FUNCTION_BLOCK "GCS7_E_Motor"	// FB 12
TITLE = Motor Control
//
//COPYRIGHT:    (C) 1996  BUHLER AG, CH-9240 UZWIL, SWITZERLAND
//
//PRODUCT:      GCS7
//
//TITLE:        Motor Control
//
//REVISION:     11  (GCPROVB)
//
//-------------------------------------------------------------------------
//
//IDENT:        AUTHOR:             DEPT:                       DATE:
//
//FB12.5.0      A. Egli             CT3                         13-Mar-2008
//              - OutpFaultReset 
//              (Software is compatible to 4.7 only GCPROVB has new revision)
//FB12.4.7      A. Egli             CT3                         04-Oct-2007
//              Interlocked Manual Mode: Use direction InOutManRev  
//FB12.4.6      A. Egli             CT3                         09-Mar-2005
//              StStopped--> StFault: Log Text 13 (not stopped)
//FB12.4.5      A. Egli             CT3                         26-Mar-2004
//              Manual Mode: Stop Motor when InHWStop or InDPFault
//FB12.4.4      A. Egli             CT3                         07-Nov-2003
//              Reset CmdOn, CmdNext when CmdOff
//FB12.4.3      A. Egli             CT3                         22-Aug-2003
//              No Start request  if InLocal
//FB12.4.2      A. Egli             CT3                         24-Jul-2003
//              Report: StStopped 
//FB12.4.1      A. Egli             CT3                         18-Jun-2003
//              Message Fault Started=Text Nr 11 
//FB12.4.0      A. Egli             CT3                         17-Jun-2002
//              New Release with one block 
//FB12.3.2      A.Egli              CT3                         22-Mai-2002
//              StStopped: Error 11: Fault stopping    
//FB12.3.1      A.Egli              CT3                         09-Nov-2001
//              Transition StStopping-->Starting in Local mode (InpFaultDev=0)    
//              Transition StStopping-->Stopped  in Local mode (InpFaultDev=1)    
//FB12.3.0      A.Egli              CT3                         28-Okt-2001
//              StCode 30: InpFaultDev=1 and InLocal=1              
//              StCode 31: InpFaultDev=1 and InLocal=0              
//FB12.2.11     A.Egli              CT3                         13-Mar-2001
//              Transition StStarting-->StFault in Local mode              
//FB12.2.10     A.Egli              CT3                         22-Jan-2001
//              Transition StStarting-->StFault after t0              
//              Interlocking PC Direct Control command with Gr.OutManualOff
//FB12.2.9      S. Kalberer         CT3                         28-Nov-2000
//              Condition for StStarting: No #tmpHeavyStartup (Netzwerk 8)      
//FB12.2.8      A. Egli             CT3                         24-Jul-2000
//              Local mode:  Transition Stopping -> Starting adapted
//FB12.2.7      S. Kalberer         CT3                         15-Mar-2000
//              Manual mode: Transition Stopping -> Starting adapted
//FB12.2.6      S. Kalberer         CT3                         02-Nov-1999
//              Count stopping time in StFault, StCode with InLocal adapted
//FB12.2E       S. Kalberer         CT3                         07-Apr-1999
//              Set outputs in StStarted Passive -> Active
//FB12.2D       A. Egli             CT3                         21-Dec-1998
//              StStopping by change speed if ParRestartDelay is true
//              Local mode: stay in StStopped if InpFaultDev = 1
//FB12.2C       A. Egli             CT3                         23-Nov-1998
//              InLocal; StStartedFdw or StStartedRev if input is set
//FB12.2B       A. Egli             CT3                         17-Jul-1998
//              Run Monitoring Time by changing speed
//FB12.2A       A. Egli             CT3                         04-Mai-1998
//              StFault = StCode 32
//FB12.1A       S. Kalberer         AEE61                       14-Jul-1997
//              1st Release in S7
//
//-------------------------------------------------------------------------
//
//PURPOSE:      MANUAL : see [MxxMAN]
//
//RESTRICTIONS: S7
//              ACCU2: Pointer to dynamic datas of the element
//              ACCU1: Pointer to parameter datas of the element
//              CmdOff, CmdOn: always active unless local mode
//
//-------------------------------------------------------------------------
//=======================================================
//Log Message: 
//------------------------------------------------------
// 0  stopped
// 2  started forward
// 5  started reverse
// 9  fault cancelled
//10  fault device
//11  fault running
//12  fault starting
//13  fault stopping
//
//=======================================================
//StCode:  State               
//------------------------------------------------------
//32 StFault+InpFaultDev=0     fault
//31 StFault+InpFaultDev=1     fault Device        (Active)
// 1 StStopped                 Stopped
//41 Stopped.HWStop            StStopped + InHWStop 
//51 Stopped.DPFault           StStopped + DPFault
//61 StStopped.FaultDev        StStopped + FaultDevice (Passiv)
// 2 StStarting                starting
// 3 StStartedFwdSlow          started forward slow
// 4 StStartedFwdFast          started forward fast
// 5 StStartedRevSlow          started reverse slow
// 6 StStartedRevFast          started reverse fast
// 7 StStopping                stopping
// 9 StStartRequest            StStopped+CmdNext
AUTHOR : EA
FAMILY : GCS7LL
NAME : Motor
VERSION : 5.0
VAR
  StCode : INT ;	//Element state code
  InEnableRev : BOOL ;	//Enable to run the element reverse
  InEnableFwd : BOOL ;	//Enable to run the element forward
  InSlow : BOOL ;	//Speed mode: 1= slow / 0= fast
  InpRunSlow : BOOL ;	//Digital input: 1= element is running slow
  InpRunFast : BOOL ;	//Digital input: 1= element is running fast
  InpRunRev : BOOL ;	//Digital input: 1= element is running reverse
  InpRunFwd : BOOL ;	//Digital input: 1= element is running forward
  InpFaultDev : BOOL ;	//Digital input: 1= overload or fault frequency converter
  CmdOff : BOOL ;	//Pulse to stop the element immediately (manual mode)
  CmdOn : BOOL ;	//Pulse to start the element immediately (manual mode)
  CmdNext : BOOL ;	//Pulse to start the element in automatic mode (see global flags)
  CmdFaultReset : BOOL ;	//Command to reset fault
  InLocal : BOOL ;	//1= Local mode (no fault by start with service switch)
  InManual : BOOL ;	//1= Manual/ 0=Automatic
  InReport : BOOL ;	//Report of all state transitions
  InSeqStop : BOOL ;	//Stop automatically after idling time
  InHWStop : BOOL ;	//HW stop is detected, no fault
  InDPFault : BOOL ;	//DP-Fault is detected, no fault
  OutIdling : BOOL ;	//Idling is active
  OutpRunSlow : BOOL ;	//Digital output to run slow
  OutpRunFast : BOOL ;	//Digital output to run fast
  OutpRunRev : BOOL ;	//Digital output to run reverse
  OutpRunFwd : BOOL ;	//Digital output to run forward
  OutpFaultReset : BOOL ;	//Reset Alarm (e.g.Softstart)
  StStopped : BOOL ;	//Element is stopped
  StStarting : BOOL ;	//Element is starting
  StStartedFwd : BOOL ;	//Element is started forward: Next element can start
  StStopping : BOOL ;	//Element is stopping
  StFault : BOOL ;	//Element has a fault
  StStartedRev : BOOL ;	//Element is started reverse: Next Element can start
  InOutManSlow : BOOL ;	//Manual speed mode: 1= slow / 0= fast
  InOutManRev : BOOL ;	//Manual direction mode: 1= reverse / 0= forward
  OutAlarmNrLog : INT ;	//Last textnumber send to log
  Par : STRUCT
   ParObjectNo : INT ;	//Is used for communication with PC, e.g. for message
   ParMsgType : INT ;	//Is used for message (translation of state)
   ParHornCode : INT ;	//Is used by horn module
   ParLogOff : BOOL ;	//Report is off
   ParManual : BOOL ;	//Manual mode without interlocking
   ParRestartDelay : BOOL ;	//No restart possible in StStopping
   Par2Speed : BOOL ;	//Element with 2 speeds
   ParHeavyStartup : BOOL ;	//Element with heavy startup
   spare45 : BOOL ;
   spare46 : BOOL ;
   OutEdgeFaultReset : BOOL ;	//Internal used
   OutDelayFault : BOOL ;	//Delay time is running: Changing speed
   OutFlagFaultDev : BOOL ;	//Flag InpFaultDev
   ParMonTime : INT ;	//After this time outputs must be equal inputs
   ParStartingTime : INT ;	//Delay time, until the element is ready to start production
   ParStoppingTime : INT ;	//Delay time, until the element has come to a standstill
   ParIdlingTime : INT ;	//Requested idling time to stop element in automatic mode
   ParDelayTime : INT ;	//Requested fault delay time by negative flag of input
   OutMonTime : INT ;	//Actual time: Monitoring
   OutTransitionTime : INT ;	//Actual time: Starting, stopping, change direction, idling
   OutDelayTime : INT ;	//Actual time: DelayTime
   InOutManPulseLen : INT ;	//Pulse length to start a the motor
  END_STRUCT ;
END_VAR
VAR_TEMP
  tmpLOGvalue : WORD ;	//LOG value
  tmpLenDyn : DINT ;
  tmpReport : BOOL ;	//Global LOG all
  tmpEnableRev : BOOL ;	//Global enable reverse
  tmpEnableFwd : BOOL ;	//Global enable forward
  tmpEnable : BOOL ;	//Global enable
  tmpSlow : BOOL ;	//Global slow speed flag
  tmpDelayOver : BOOL ;	//Delay time is over
  tmpMonOver : BOOL ;	//Monitoring time is over
  tmpTimeClear : BOOL ;	//Delay- and monitoring time must be cleared
  tmpStop : BOOL ;	//States to clear outputs
  tmpInpOutpDiff : BOOL ;	//Inpputs ar different to outputs
  tmpInpFault : BOOL ;	//Fault variable
  tmpInpRunSlow : BOOL ;	//Variable to simulate InpRunSlow
  tmpHeavyStartup : BOOL ;	//Any element is starting with HeavyStartup
  tmpLocal : BOOL ;
  tmpFaultDelayDone : BOOL ;
  tmpStarted : BOOL ;
END_VAR
BEGIN
NETWORK
TITLE =  Start Global
      L     34;
      T     #tmpLenDyn;	//--> Len dynamic data in byte
NETWORK
TITLE = PC Control
//=== Test Object number =====================
      L     "SYS_DirectCtrlDB".PC.ObjectNo;	//PCControl.ObjectNo
      L     #Par.ParObjectNo;	//Input ObjectNo
      <>I;
      JC    Ctrl;
//=== Test OType      ========================
      L     1012;	//Input object type
      L     "SYS_DirectCtrlDB".PC.ObjectType;	//PCControl.ObjectType
      <>I;
      JC    Ctrl;
//=== Test Handshake =========================
      A     "SYS_DirectCtrlDB".PC.Hsk.FExamine;	// Handshake.FExamine
      JC    pExa;
      A     "SYS_DirectCtrlDB".PC.Hsk.FDefineCmd;	// Handshake.FDefineCmd
      JC    pCmd;
      A     "SYS_DirectCtrlDB".PC.Hsk.FDefinePara;	// Handshake.FDefinePara
      JC    pPar;
pIni: L     2;	// FcInit
      UC    "SYS_DirectCtrl";
      JU    Ctrl;
// Write parameter 
pPar: LAR1  P#DBX 58.0;
      L     P##Par;
      L     DW#16#FFFFF;
      AD;
      +AR1;
      L     DBW [AR1,P#8.0];
      T     #Par.ParMonTime;
      L     DBW [AR1,P#10.0];
      T     #Par.ParStartingTime;
      L     DBW [AR1,P#12.0];
      T     #Par.ParStoppingTime;
      L     DBW [AR1,P#14.0];
      T     #Par.ParIdlingTime;
      L     DBW [AR1,P#16.0];
      T     #Par.ParDelayTime;
// Write new commands from PC to Interface object
pCmd: A     "SYS_DirectCtrlDB".PC.Cmd1[6];	// CmdManSlowOn
      AN    "GCS7_Gr_OutManualOff";	//Global.OutManualOff  [2.10]
      S     #InOutManSlow;
      A     "SYS_DirectCtrlDB".PC.Cmd1[7];	// CmdManRevOn;
      AN    "GCS7_Gr_OutManualOff";	//Global.OutManualOff  [2.10]
      S     #InOutManRev;
      A     "SYS_DirectCtrlDB".PC.Cmd1[8];	// CmdOff
      AN    "GCS7_Gr_OutManualOff";	//Global.OutManualOff  [2.10]
      S     #CmdOff;
      A     "SYS_DirectCtrlDB".PC.Cmd1[9];	// CmdOn
      AN    "GCS7_Gr_OutManualOff";	//Global.OutManualOff  [2.10]
      S     #CmdOn;
      A     "SYS_DirectCtrlDB".PC.Cmd1[10];	// CmdNext
      S     #CmdNext;
      A     "SYS_DirectCtrlDB".PC.Cmd1[11];	// CmdFaultReset
      S     #CmdFaultReset;
      A     "SYS_DirectCtrlDB".PC.Cmd1[13];	// CmdManualOn
      S     #InManual;
      A     "SYS_DirectCtrlDB".PC.Cmd1[14];	// CmdReportOn
      S     #InReport;
      A     "SYS_DirectCtrlDB".PC.Cmd2[6];	// CmdManSlowOff
      R     #InOutManSlow;
      A     "SYS_DirectCtrlDB".PC.Cmd2[7];	// CmdManRevOff;
      R     #InOutManRev;
      A     "SYS_DirectCtrlDB".PC.Cmd2[13];	// CmdManualOff
      R     #InManual;
      A     "SYS_DirectCtrlDB".PC.Cmd2[14];	// CmdReportOff
      R     #InReport;
      AN    "SYS_DirectCtrlDB".PC.Cmd1[1];	// CmdOnTickFwd
      O     "GCS7_Gr_OutManualOff";	//Global.OutManualOff
      JC    pIni;
      L     "SYS_DirectCtrlDB".PC.Cmd3;	// "SYS_PCControl".PC.Cmd3
      T     #Par.InOutManPulseLen;
      JU    pIni;
pExa: TAR2;	// Address Dynamic datas
      T     "SYS_DirectCtrlDB".GC.InDynAddr;	// -->PCControl.GC.InDynAddr
      L     #tmpLenDyn;	// Length Dynamic datas
      T     "SYS_DirectCtrlDB".GC.InDynLen;	// -->PCControl.GC.InDynLen
      L     0;
      T     "SYS_DirectCtrlDB".GC.InParaAddr;	// -->PCControl.GC.InParaAddr
      T     "SYS_DirectCtrlDB".GC.InParaLen;	// -->PCControl.GC.InParaLen
      L     1;	// Code FcExamine
      UC    "SYS_DirectCtrl";
      L     11;	//Revision
      T     "SYS_DirectCtrlDB".GC.Revision;
NETWORK
TITLE =  All State Init
//===Clear tmp Variable, when nessecary
Ctrl: CLR;
      =     #tmpTimeClear;
//===Global Group Orders===
      A     "GCS7_Gr_OutManualOn";	//Global.OutManualOn
      S     #InManual;
      A     "GCS7_Gr_OutManualOff";	//Global.OutManualOff
      R     #InManual;
      A     #InManual;
      S     "GCS7_Gr_InManual";	//Global.InManualMode
      AN    #InManual;
      A     #InLocal;
      =     #tmpLocal;
//---Report is on---
      O     "GCS7_Gr_OutReportAll";	//---Global OutReportAll
      O     #InReport;
      =     #tmpReport;
//---Heavy Startup---
      A     "GCS7_Gr_InHeavyStartup";	//---Global InHeavyStartup
      A     #Par.ParHeavyStartup;
      =     #tmpHeavyStartup;
//===Global Enable and Speed===
      A     #CmdOff;	//[4.4]
      R     #CmdOn;	//[4.4]
      R     #CmdNext;	//[4.4]
//---Enable / Manual No Interlocking Mode---
      AN    #InManual;
      JC    AUT;
      A(;	//[4.5]
      A     #InEnableFwd;
      AN    #InOutManRev;	//[4.7]
      AN    #Par.ParManual;
      O;
      AN    #InOutManRev;
      A     #Par.ParManual;
      );	//[4.5]
      AN    #InHWStop;	//[4.5]
      AN    #InDPFault;	//[4.5]
      =     #tmpEnableFwd;
      A(;	//[4.5]
      A     #InEnableRev;
      A     #InOutManRev;	//[4.7]
      AN    #Par.ParManual;
      O;
      A     #InOutManRev;
      A     #Par.ParManual;
      );	//[4.5]
      AN    #InHWStop;	//[4.5]
      AN    #InDPFault;	//[4.5]
      =     #tmpEnableRev;
//---Speed / Manual No Interlocking Mode---
      A     #InOutManSlow;
      ON    #Par.Par2Speed;
      =     #tmpSlow;
      JU    ENAB;
//---Enable / Automatic Interlocking Mode---
AUT:  A     #InEnableFwd;
      AN    #InHWStop;
      AN    #InDPFault;
      AN    #InLocal;
      =     #tmpEnableFwd;
      A     #InEnableRev;
      AN    #InHWStop;
      AN    #InDPFault;
      AN    #InLocal;
      =     #tmpEnableRev;
//---Speed / Automatic Interlocking Mode---
      A     #InSlow;
      ON    #Par.Par2Speed;
      =     #tmpSlow;
//---Enable / HardwareStop---
ENAB: X     #tmpEnableFwd;	//---Global Enable
      X     #tmpEnableRev;
      =     #tmpEnable;
//---For one speed, no Inp nessecary: Simulate InpRunSlow
      AN    #Par.Par2Speed;
      A     #OutpRunSlow;
      =     #tmpInpRunSlow;
// Check Input different to Output
      A     #InpRunFwd;
      X     #OutpRunFwd;
      O(;
      A     #InpRunRev;
      X     #OutpRunRev;
      );
      O(;
      A     #InpRunFast;
      X     #OutpRunFast;
      );
      O(;
      O     #InpRunSlow;
      O     #tmpInpRunSlow;
      X     #OutpRunSlow;
      );
      =     #tmpInpOutpDiff;
//---Both Inputs or InpFaultDevice active
      A     #InpRunFwd;	// local StStarting
      A     #InpRunRev;
      O;
      A     #InpRunSlow;	// local StStarting
      A     #InpRunFast;
      =     #tmpInpFault;
NETWORK
TITLE = Start as Pulse
      AN    #tmpEnable;
      ON    #InManual;
      O     #CmdOff;
      JC    STP1;
      L     0;
      L     #Par.InOutManPulseLen;
      >=I;
      JC    STP2;
      S     #CmdOn;
      AN    "GCS7_Gr_OutTick200ms";	// Decrement all 200ms
      JC    STP2;
      +     -2;
      T     #Par.InOutManPulseLen;
      L     0;
      >I;
      JC    STP2;
      S     #CmdOff;
STP1: L     0;
      T     #Par.InOutManPulseLen;
STP2: NOP   0;
NETWORK
TITLE = Fault delay time: ParDelayTime 
//Test or Running delay time ====================
//---Condition for Delay Fault
      AN    #tmpInpOutpDiff;
      AN    #InpFaultDev;
      O     #InHWStop;
      O     #InDPFault;
      JC    TFDO;
      A     #StStartedFwd;
      O     #StStartedRev;
      AN    #Par.OutDelayFault;
      O     #StStopped;
      A     #tmpInpOutpDiff;
      O     #InpFaultDev;
      JC    TFF1;
TFDO: R     #tmpFaultDelayDone;
      L     0;
      T     #Par.OutDelayTime;
      JU    TFF0;
TFF1: AN    "GCS7_Gr_OutTick200ms";	// Decrement all 200ms
      L     #Par.OutDelayTime;
      JC    TFF3;
      +     2;
TFF3: T     #Par.OutDelayTime;
      L     #Par.ParDelayTime;
      >=I;
      =     #tmpFaultDelayDone;
      JCN   TFF0;
      T     #Par.OutDelayTime;
TFF0: NOP   0;
NETWORK
TITLE = States
      O     #StStartedFwd;
      O     #StStartedRev;
      =     #tmpStarted;
      A     #StStopped;	//===State machine===
      JC    S0;
      O     #StStartedFwd;
      O     #StStartedRev;
      JC    S2;
      A     #StStopping;
      JC    S3;
      A     #StStarting;
      JC    S1;
      A     #StFault;
      JC    S4;
      S     #StStopped;	//Initialise: goto StStopped
NETWORK
TITLE = StStopped
//---Condition for StFault
S0:   A     #tmpFaultDelayDone;	// [4.0]
      O     #tmpInpFault;
      AN    #tmpLocal;	//2D:
      JC    S0S4;
//---Condition for StStarting: local
      AN    #tmpLocal;
      JC    S0J1;
      X     #InpRunFwd;
      X     #InpRunRev;
      JC    S0S1;
      JU    SAVE;
//---Condition for StStopped
S0J1: O     #CmdOff;
      ON    #tmpEnable;
      JC    SAVE;
//---Condition for StStarting: automatic
      O     #CmdNext;
      O     #CmdOn;
      AN    #InManual;
      AN    #InSeqStop;
      AN    #tmpHeavyStartup;
      JC    S0S1;
//---Condition for StStarting: manual 
      A     #InManual;
      A     #CmdOn;
      JCN   SAVE;
//---Transition -> StStarting
S0S1: R     #StStopped;
      JU    xxS1;
//---Transition -> StFault
S0S4: R     #StStopped;
      R     #tmpEnable;	//[4.6]
      JU    xxS4;
NETWORK
TITLE = StStarting
//== Any transition to StStarting
xxS1: SET;
      S     #StStarting;
      L     #Par.ParMonTime;	// Set actual vaule of timer
      T     #Par.OutMonTime;
      L     #Par.ParStartingTime;
      T     #Par.OutTransitionTime;
      A     #tmpLocal;	// No output set in local mode
      JC    SAVE;
      A     #Par.ParHeavyStartup;	// Set Global InHeavyStartup
      S     "GCS7_Gr_InHeavyStartup";
      A     #tmpEnableFwd;	// Set direction
      =     #OutpRunFwd;
      A     #tmpEnableRev;
      =     #OutpRunRev;
      A     #tmpSlow;	// Set speed
      =     #OutpRunSlow;
      NOT;
      =     #OutpRunFast;
      JU    SAVE;
//== Logic ====
//---Condition for StFault
S1:   A     #tmpInpFault;
      O     #tmpFaultDelayDone;	// [4.0]
      AN    #tmpLocal;
      JC    S1S4;
//---Condition for StStopped  local mode
      AN    #tmpLocal;
      JC    S11;
      A     #InpRunRev;
      XN    #InpRunFwd;
      JC    S1S3;
      JU    S12;
//---Condition for StStopped  other modes
S11:  ON    #tmpEnable;
      O     #CmdOff;
      O;
      A     #InSeqStop;
      AN    #InManual;
      O;
      AN    #OutpRunFwd;
      AN    #OutpRunRev;
      JC    S1S3;
//---Condition for StStarting
S12:  AN    "GCS7_Gr_OutTick200ms";
      L     #Par.OutTransitionTime;	// Set Timer 
      JC    S13;
      L     #Par.OutMonTime;
      +     -2;
      T     #Par.OutMonTime;
      L     #Par.OutTransitionTime;
      +     -2;
      T     #Par.OutTransitionTime;
S13:  L     0;
      <=I;	//---Condition for StStarted
      =     #tmpDelayOver;	// Starting time over
      A     #tmpDelayOver;	// Started forward
      A     #tmpEnableFwd;
      AN    #tmpInpOutpDiff;
      O;
      A     #tmpDelayOver;	// Started forward local  
      A     #InpRunFwd;
      A     #tmpLocal;
      JC    S1S2;
      A     #tmpDelayOver;	// Started reverse
      A     #tmpEnableRev;
      AN    #tmpInpOutpDiff;
      O;
      A     #tmpDelayOver;	// Started reverse local  
      A     #InpRunRev;
      A     #tmpLocal;
      JC    S15;
      L     #Par.OutMonTime;	//---Condition for StFault
      L     0;	// Monitoring time over
      <=I;
//      U     #tmpDelayOver; // Starting time over [2.10]
      AN    #tmpLocal;	//[2.11]
      A     #tmpInpOutpDiff;	// Inp not equal Outp
      JC    S1S4;
      JU    SAVE;
S1S2: R     #StStarting;	//---Transition -> StStartedFwd
      S     #StStartedFwd;
      S     #tmpTimeClear;	// Reset actual timer value
      A     #tmpHeavyStartup;	// Clear Global InHeavyStartup
      R     "GCS7_Gr_InHeavyStartup";
      JU    LOG1;
S15:  R     #StStarting;	//---Transition -> StStartedRev
      S     #StStartedRev;
      S     #tmpTimeClear;	// Reset actual timer value
      A     #tmpHeavyStartup;	// Clear Global InHeavyStartup
      R     "GCS7_Gr_InHeavyStartup";
      JU    LOG1;
//---Transition -> StStopping
S1S3: R     #StStarting;
      A     #tmpHeavyStartup;	// Clear Global InHeavyStartup
      R     "GCS7_Gr_InHeavyStartup";
      JU    xxS3;
//---Transition -> StFault
S1S4: R     #StStarting;
      A     #tmpHeavyStartup;	// Clear Global InHeavyStartup
      R     "GCS7_Gr_InHeavyStartup";
      JU    xxS4;
NETWORK
TITLE = StStarted
S2:   A     #tmpInpFault;	//---Condition for StFault
      O     #tmpFaultDelayDone;	// [4.0]
      AN    #tmpLocal;
      JC    S2S4;
//---Condition for StStopping: local mode
      AN    #tmpLocal;
      JC    S2J1;	// no speed changing and no idling 
      A     #StStartedFwd;	// Input Fwd goes off
      AN    #InpRunFwd;
      O;
      A     #StStartedRev;	// Input Rev goes off
      AN    #InpRunRev;
      JC    S2S3;
      JU    SAVE;
//---Condition for StStopping: autmatic
S2J1: A     #Par.Par2Speed;	//[Rel 2D -->
      A     #Par.ParRestartDelay;
      A     #tmpSlow;
      AN    #OutpRunSlow;
      O;
      A     #Par.Par2Speed;
      A     #Par.ParRestartDelay;
      AN    #tmpSlow;
      A     #OutpRunSlow;
      JC    S2S3;	// Condition for StStoppping  Rel 2D <--]
      ON    #tmpEnable;	// other modes
      O     #CmdOff;
      O;
      A     #OutpRunFwd;	// Change direction: Fwd --> Rev
      A     #tmpEnableRev;
      O;
      A     #OutpRunRev;	// Change direction: Rev --> Fwd
      A     #tmpEnableFwd;
      JC    S2S3;
//2E:---Condition for StStarted: set direction outputs
      A     #tmpEnableFwd;
      =     #OutpRunFwd;
      A     #tmpEnableRev;
      =     #OutpRunRev;
//---Condition for StStarted: speed changing
      A     #OutpRunSlow;
      AN    #tmpSlow;
      A     #Par.Par2Speed;	// Doubt only one speed
      AN    #Par.OutDelayFault;
      O;
      A     #OutpRunFast;	//---Condition for StStarted: speed changing
      A     #tmpSlow;
      A     #Par.Par2Speed;	// Doubt only one speed
      AN    #Par.OutDelayFault;
      JCN   S2F1;
      S     #Par.OutDelayFault;
      L     #Par.ParMonTime;
      L     #Par.ParDelayTime;
      <=I;
      JC    S2F2;
      L     #Par.ParMonTime;
S2F2: T     #Par.OutMonTime;
      JU    SAVE;
S2F1: A     #InpRunSlow;
      O     #InpRunFast;
      ON    #Par.Par2Speed;	// Doubt only one speed
      JC    S2J2;
      A     #tmpSlow;	// Set speed
      =     #OutpRunSlow;
      NOT;
      =     #OutpRunFast;
//Test or Running delay time ====================
S2J2: A     #tmpInpOutpDiff;	//---Condition for Delay Fault
      A     #Par.OutDelayFault;	// Set OutDelayFault Bit
      JC    S2T1;
      A     #InpRunFast;
      O     #InpRunSlow;
      ON    #Par.Par2Speed;	// Doubt only one speed
      A     #Par.OutDelayFault;
      JCN   S2J3;	// Check Idling
      R     #Par.OutDelayFault;
      S     #tmpTimeClear;
      JU    SAVE;
S2T1: AN    "GCS7_Gr_OutTick200ms";	// Decrement all 200ms
      L     #Par.OutMonTime;
      JC    S2T3;
      +     -2;
      T     #Par.OutMonTime;
S2T3: L     0;
      <=I;
      R     #Par.OutDelayFault;
      JCN   SAVE;
      A     #tmpEnable;	// Condition for StFault
      JC    S2S4;
      JU    S2S3;	// Condition for StStoppping
//---Idling time ----------------------
S2J3: O     #InSeqStop;
      ON    #OutIdling;	// Condition to reset Idling-Time
      JC    S2I1;
      R     #OutIdling;
      S     #tmpTimeClear;	// Reset actual timer value
      JU    SAVE;
S2I1: ON    #InSeqStop;	// Idling time active ?
      O     #InManual;
      JC    SAVE;
      A     #OutIdling;
      JC    S2I2;
      S     #OutIdling;	// Preset Idling Time
      L     #Par.ParIdlingTime;
      T     #Par.OutTransitionTime;
S2I2: AN    "GCS7_Gr_OutTick200ms";	// Set Idling Time
      L     #Par.OutTransitionTime;
      JC    S2I3;
      +     -2;
      T     #Par.OutTransitionTime;
S2I3: L     0;
      >I;	// Idling time over
      JC    SAVE;
S2S3: R     #StStartedFwd;	//---Transition -> StStopping
      R     #StStartedRev;
      R     #Par.OutDelayFault;
      JU    xxS3;
S2S4: R     #StStartedFwd;	//---Transition -> StFault
      R     #StStartedRev;
      R     #Par.OutDelayFault;
      R     #OutIdling;
      JU    xxS4;
NETWORK
TITLE = StStopping
//===Any transition to StStopping
xxS3: SET;
      S     #StStopping;
      R     #OutIdling;
      L     #Par.ParMonTime;	// Set monitoring time
      T     #Par.OutMonTime;
      L     #Par.ParStoppingTime;	// Set stopping time
      T     #Par.OutTransitionTime;
      JU    SAVE;
//===Logic =======================
//---Condition for StFault
S3:   A     #tmpInpFault;
      O     #tmpFaultDelayDone;	// [4.0]
      AN    #tmpLocal;	//[2.8] 
      JC    S3S4;
//---Condition for StStarting in InLocal
//[3.1]      U     #tmpInpFault                //[2.8]
//[3.1]      U     #tmpLocal                   //[2.8] 
//[3.1]      SPB   SAVE                        //[2.8]  
      X     #InpRunFwd;	//[2.8]
      X     #InpRunRev;	//[2.8]
      AN    #tmpInpFault;	//[3.1]
      A     #tmpLocal;	//[2.8] 
      JC    S3S1;	//[2.8] Transition -> StStarting 
//---Condition for StStarting: no Restart
      A     #Par.ParRestartDelay;
      O     #tmpHeavyStartup;	//[2.9]
      JC    S3J2;
      O     #CmdNext;	// automatic StStarting
      O     #CmdOn;
      AN    #InManual;
      AN    #InSeqStop;
      A     #tmpEnable;
      AN    #tmpLocal;	//[3.1] 
      JC    S3S1;
      A     #InManual;	// manual StStarting
      A     #CmdOn;
      A     #tmpEnable;	// [2.7]
      JC    S3S1;
//---Condition for StStopping
S3J2: AN    "GCS7_Gr_OutTick200ms";
      L     #Par.OutTransitionTime;	// Set Timer 
      JC    S3J3;
      L     #Par.OutMonTime;	//---Condition for StStopped
      +     -2;	// Set actual timer
      T     #Par.OutMonTime;
      L     #Par.OutTransitionTime;
      +     -2;
      T     #Par.OutTransitionTime;
S3J3: L     0;
      <=I;	// Stopping time over
      =     #tmpDelayOver;
      A     #tmpDelayOver;	// Stopped
      AN    #tmpInpOutpDiff;	// Inp equal Outp
      JC    S3S0;
      L     #Par.OutMonTime;
      L     0;	// Monitoring time over
      <=I;
      =     #tmpMonOver;
      A     #tmpMonOver;
      A     #tmpDelayOver;	// Stopping time over
      AN    #tmpInpOutpDiff;	// Inp equal Outp
      JC    S3S0;
      A     #tmpMonOver;	//---Condition for StFault
      A     #tmpInpOutpDiff;
      O;
      A     #tmpMonOver;
      A     #tmpDelayOver;
      A     #tmpInpOutpDiff;
      JCN   SAVE;
//---Transtition -> StFault
S3S4: R     #StStopping;
      JU    xxS4;
//---Transition -> StStarting
S3S1: R     #StStopping;
      JU    xxS1;
//---Transition -> StStopped
S3S0: R     #StStopping;
      S     #StStopped;
      S     #tmpTimeClear;	// Reset actual timer value
      JU    LOG1;
NETWORK
TITLE =  StFault
// Any transiton to Fault  
xxS4: SET;
      S     #StFault;
      S     "GCS7_Gr_InFaultFlag";	// Global.InFaultFlag
//    S     #tmpTimeClear               // Reset actual timer value
      CALL  "SYS_Horn_Code" (
           FcCode                   := 1,
           ParObjectType            := 1012,
           ParObjectNo              := #Par.ParObjectNo,
           ParHornCode              := #Par.ParHornCode);
      L     0;	//2.6
      T     #Par.OutMonTime;
      L     #Par.ParStoppingTime;
      T     #Par.OutTransitionTime;
      SET;
S4S4: JU    LOG4;
//===logic
S4:   L     0;	//---Condition to count stopping time
      L     #Par.OutTransitionTime;	// Set Timer 
      >=I;
      ON    "GCS7_Gr_OutTick200ms";
      JC    S4J1;
      +     -2;
      T     #Par.OutTransitionTime;
S4J1: A     #InpFaultDev;
      A     #tmpFaultDelayDone;	// [4.0]
      AN    #tmpLocal;
      FP    #Par.OutFlagFaultDev;
      JC    S4S4;
      AN    #CmdFaultReset;	//---Condition for StFault
      AN    "GCS7_Gr_OutFaultReset";	// OutFaultReset
      AN    #tmpLocal;
      JC    SAVE;
      A     #InpFaultDev;	//---Condition for StFault with LOG
      O     #tmpInpFault;	// MessageClass Error Fault stopping
      O     #tmpInpOutpDiff;
      AN    #tmpLocal;
      JC    S4S4;
      R     #StFault;	//---Transition -> StStopping
      S     #StStopping;
      R     #OutIdling;
      L     #Par.ParMonTime;	// Set monitoring time
      T     #Par.OutMonTime;
      JU    LOG9;
NETWORK
TITLE = LOG Message
//LOG transition to StStopped,StStartedXxx
LOG1: AN    #tmpReport;	// ReportAll?
      JC    SAVE;
      A     #StStartedFwd;
      L     B#(4, 2);	// MessageClass Info started fwd
      JC    LOG;
      A     #StStartedRev;
      L     B#(4, 5);	// MessageClass Info started rev
      JC    LOG;
      A     #StStopped;
      L     B#(4, 0);	// MessageClass Info stopped
      JC    LOG;	// [4.2]
      JU    SAVE;
//LOG transition to fault
LOG4: A     #InpFaultDev;
      =     #Par.OutFlagFaultDev;	//[4.0]
      L     B#(1, 10);	// MessageClass Error fault device
      JC    LOG;
      A     #tmpStarted;
      L     B#(1, 11);	// MessageClass Error fault started
      JC    LOG;
      AN    #tmpEnable;	//Fault Stopping
      L     B#(1, 13);
      JC    LOG;
      L     B#(1, 12);	// MessageClass Error fault starting
      JU    LOG;
//Log fault cancelled
LOG9: L     B#(3, 9);	// MessageClass Operater "fault cancelled"
LOG:  A     #Par.ParLogOff;	//---Set LOG Message
      JC    SAVE;
      T     #tmpLOGvalue;
      L     W#16#FF;
      AW;
      T     #OutAlarmNrLog;
      CALL  "GCS7_LogConvert" (
           ObjectNo                 := #Par.ParObjectNo,
           MsgType                  := #Par.ParMsgType,
           ClassMsgTxt              := #tmpLOGvalue,
           OType                    := 1012);	// LOG Message Converter / Entry / Contains Class and TextNo
NETWORK
TITLE = State Code
//--Stopped, Substate ---
SAVE: AN    #StStopped;
      JC    STC2;
      L     41;	//Code: StStopped.HWStop
      A     #InHWStop;
      JC    STC9;
      L     51;	//Code: StStopped.DPFault
      A     #InDPFault;
      JC    STC9;
      A     #InpFaultDev;	// 
      L     30;	//Code: StStopped.InpFaultDev
      JC    STC9;	// 
      A     #CmdNext;
      AN    #tmpLocal;	//[4.3]
      L     9;	// Code: starting requested
      JC    STC9;
      L     1;	// Code: stopped
      JC    STC9;
//--------------------
STC2: A     #StStarting;
      L     2;	// Code: starting
      JC    STC9;
      AN    #StStartedFwd;
      JC    STC3;
      L     3;	// 2.6 Code: started forward slow
      A     #InLocal;
      A     #InpRunSlow;
      O     #OutpRunSlow;
      ON    #Par.Par2Speed;
      JC    STC9;
      L     4;	// Code: started forward fast
      JU    STC9;
//--------------------
STC3: AN    #StStartedRev;
      JC    STC4;
      L     5;	// 2.6: Code: started reverse slow
      A     #InLocal;
      A     #InpRunSlow;
      O     #OutpRunSlow;
      ON    #Par.Par2Speed;
      JC    STC9;
      L     6;	// Code: started reverse fast
      JU    STC9;
//--------------------
STC4: A     #StStopping;
      L     7;	// Code: stopping
      JC    STC9;
      A     #InpFaultDev;	// [3.0]
      L     31;	// [3.0]
      JC    STC9;	// [3.0]
      L     32;	// Code: fault
STC9: L     #StCode;	// Old state code
      TAK;
      T     #StCode;	// Save state code
      <>I;
      L     3;	// Load code for CBit methode
      CC    "SYS_CBitCtrl";
NETWORK
TITLE = Global End
      A     #CmdFaultReset;	//[5.0]
      S     #Par.OutEdgeFaultReset;	//[5.0]
      A     "GCS7_Gr_OutTick1s";	//[5.0]
      R     #OutpFaultReset;	//[5.0]
      A     "GCS7_Gr_OutTick1s";	//[5.0]
      A     #Par.OutEdgeFaultReset;	//[5.0]
      R     #Par.OutEdgeFaultReset;	//[5.0]
      S     #OutpFaultReset;	//[5.0]
//---Clear all commands
      CLR;
      =     #CmdOn;
      =     #CmdOff;
      =     #CmdNext;
      =     #CmdFaultReset;
      O     #StStopped;	//---Reset Hardware Outputs
      O     #StStopping;
      O     #StFault;
      =     #tmpStop;
      ON    #tmpEnableFwd;	// Output Forward
      O     #tmpStop;
      R     #OutpRunFwd;
      ON    #tmpEnableRev;	// Output Reverse
      O     #tmpStop;
      R     #OutpRunRev;
      ON    #tmpSlow;	// Output Slow
      O     #tmpStop;
      R     #OutpRunSlow;
      O     #tmpSlow;	// Output Fast
      O     #tmpStop;
      R     #OutpRunFast;
//--Output for group 
      AN    #InLocal;
      O     #InManual;
      A     #InDPFault;
      S     "GCS7_Gr_InDPFault";
      AN    #InLocal;
      O     #InManual;
      A     #InHWStop;
      S     "GCS7_Gr_InHWStop";
//---Reset actual timer values
      AN    #tmpTimeClear;
      BEC;
      L     0;
      T     #Par.OutMonTime;
      T     #Par.OutTransitionTime;
END_FUNCTION_BLOCK

FUNCTION_BLOCK "GCS7_E_ValveControl"	// FB 13
TITLE = ValveControl
//  
//COPYRIGHT:    (C) 1996  BUHLER AG, CH-9240 UZWIL, SWITZERLAND
//
//PRODUCT:      GCS7
//
//TITLE:        Valve Control with Limit Switch (VLS)
//
//-------------------------------------------------------------------------
//
//IDENT:        AUTHOR:             DEPT:                       DATE:
//
//FB13.4.6      A. Egli             CT3                         02-Dec-2004
//              PCD:Ignor CmdLN, CmdHN as con M12.4=1
//FB13.4.5      A. Egli             CT3                         26-Nov-2004
//              ParDelayTime always used also for InpFaultDev
//FB13.4.4      A. Egli             CT3                         28-Jun-2004
//              Init state after Download is StNoPosition
//FB13.4.3      A. Egli             CT3                         04-Sep-2003
//              InStopCTime, StCode=12, StCode=14
//FB13.4.2      A. Egli             CT3                         04-Sep-2003
//              Message Text: Fault opening =12, fault closing=11
//FB13.4.1      A. Egli             CT3                         16-Jun-2003
//              Store text number, when calling FC4 
//FB13.4.0      A. Egli             CT3                         17-Jun-2002
//              New Release with one block 
//FB13.2.8      A. Egli             CT3                         16-Mar-2002
//              Set minimum MonTime =0.3s
//FB13.2.7      A. Egli             CT3                         03-Jul-2001
//              Transition during fault delay time is running
//FB13.2.6      S. Kalberer         CT3                         30-May-2000
//              Local mode: InpLN+InpHN -> StNoPosition
//FB13.2.5      S. Kalberer         CT3                         15-Mar-2000
//              PulseValve: change direction with CmdLN/CmdHN corrected
//FB13.2.4      S. Kalberer         CT3                         25-Nov-1999
//              PulseValve: StopAndGo corrected
//FB13.2D       A. Egli             CT3                         11-Oct-1999
//              Remove flag 12.2 (Gr.OutNext)
//FB13.2C       S. Kalberer         CT3                         05-Mar-1999
//              Interlocked Manual Mode: StHN->StLN if InEnableHN=0
//FB13.2B       A. Egli             CT3                         09-Dec-1998
//              Automatic Fault reset if InLocal
//FB13.2A       A. Egli             CT3                         04-Mai-1998
//              StFault = StCode 32
//FB13.1B       A. Egli             AEE61                       4-Nov-1997
//              ParManual
//FB13.1A       S. Kalberer         AEE61                       4-Jul-1997
//              1st Release in S7
//
//-------------------------------------------------------------------------
//
//PURPOSE:      MANUAL : see [VLSxxMAN]
//
//RESTRICTIONS: S7
//              ACCU2: Pointer to dynamic datas of the element
//              ACCU1: Pointer to parameter datas of the element
//
//-------------------------------------------------------------------------
//=======================================================
//Log Message: 
//------------------------------------------------------
// 0  LN
// 2  HN
// 9  fault cancelled
//10  fault device
//11  fault LN
//12  fault HN
//13  fault no position
//
//=======================================================
//StCode:  State               
//------------------------------------------------------
//32   StFault                 
// 1   StLN                    
//41   StLN.HWStop             StLN + InHWStop
//51   StLN.DPFault            StLN + InDPFault
// 2   StCtoHN                 
//12   StCtoHN                 StCtoHN + InStopCTime
// 3   StHN                    
//43   StHN.HWStop             StHN + InHWStop
//53   StHN.DPFault            StHN + InDPFault
// 4   StCtoLN                 
//14   StCtoLN                 StCtoLN + InStopCTime
// 5   StNoPosition            
//45   StNoPosition.HWStop     StNoPosition + InHWStop
//55   StNoPosition.DPFault    StNoPosition + InDPFault
//
//
AUTHOR : EA
FAMILY : GCS7LL
NAME : VLS
VERSION : 4.6
VAR
  StCode : INT ;	//Element state code
  InEnableLN : BOOL ;	//Target position is LN
  InEnableHN : BOOL ;	//Target position is HN
  InStopCTime : BOOL ;	//Stop Monitoring Time in State StCToLN and StCToHN
  spare0203 : BOOL ;
  spare0204 : BOOL ;
  InpLN : BOOL ;	//Digital input: limit switch low  position (closed)
  InpHN : BOOL ;	//Digital input: limit switch high position (open)
  InpFaultDev : BOOL ;	//Digital input: fault device
  CmdLN : BOOL ;	//Pulse to set position LN (manual mode)
  CmdHN : BOOL ;	//Pulse to set position HN (manual mode)
  CmdNext : BOOL ;	//Open next element
  CmdFaultReset : BOOL ;	//Command to reset fault
  InLocal : BOOL ;	//1= Local mode (no fault by start with service switch)
  InManual : BOOL ;	//1= Manual/ 0= Automatic
  InReport : BOOL ;	//Report of all state transition
  InSeqStop : BOOL ;	//Stop automatically after idling time
  InHWStop : BOOL ;	//HW stop is detected, no fault
  InDPFault : BOOL ;	//DP-Fault is detected, no fault
  OutIdling : BOOL ;	//Idling time is running
  OutDelayFault : BOOL ;	//Delay time is running
  OutMonFault : BOOL ;	//Monitoring time is running
  OutpLN : BOOL ;	//Digital output: valve low  position (closed)
  OutpHN : BOOL ;	//Digital output: valve high position (open)
  spare0407 : BOOL ;
  StLN : BOOL ;	//Element is in position LN
  StCtoHN : BOOL ;	//Changing to position HN
  StHN : BOOL ;	//Element is in position HN
  StCtoLN : BOOL ;	//Changing to position LN
  StFault : BOOL ;	//Element has a fault (time-out by positioning)
  StNoPosition : BOOL ;	//Element is not in a final position (only in local mode)
  OutAlarmNrLog : INT ;	//Last textnumber send to log
  Par : STRUCT
   ParObjectNo : INT ;	//Is used for communication with PC, e.g. for message
   ParMsgType : INT ;	//Is used for message (translation of state)
   ParHornCode : INT ;	//Is used by horn module
   ParLogOff : BOOL ;	//Report is off
   ParManual : BOOL  := TRUE;	//No interlocking in manual mode
   ParPulseValve : BOOL ;	//Valves with pulse signal
   ParContValve : BOOL ;	//Valves with continuous signal
   ParManualFlap : BOOL ;	//Manual flap, no valves
   ParMonTime : INT ;	//After this time the element mus be in final position
   ParPulseTimeHN : INT ;	//Delay time, if arrive the position HN
   ParPulseTimeLN : INT ;	//Delay time, if arrive the position LN
   ParIdlingTime : INT ;	//Requested idling time to close valve in automatic mode
   ParDelayTime : INT ;	//Requested fault delay time by negative flag of input
   OutMonTime : INT ;	//Actual time: Monitoring
   OutTransitionTime : INT ;	//Actual time: Change to LN or HN
   OutDelayTime : INT ;	//Actual time: DelayTime
   InOutManPulseLen : INT ;	//Pulse length to Move to HN
  END_STRUCT ;
END_VAR
VAR_TEMP
  tmpLOGvalue : WORD ;	//LOG value
  tmpLenDyn : DINT ;
  tmpReport : BOOL ;	//Global LOG all
  tmpEnable : BOOL ;	//Global enable
  tmpInpOk : BOOL ;	//Input ok variable
  tmpDelayOver : BOOL ;	//Delay time is over
  tmpDelayClear : BOOL ;	//Delay time must be cleared
  tmpMonFault : BOOL ;	//Global monitor fault
  tmpMonOver : BOOL ;	//Monitoring time over
  tmpMonClear : BOOL ;	//Monitoring time must be cleared
  tmpNoMon : BOOL ;	//Monitoring not active
  tmpManStopGo : BOOL ;	//Condition for StopAndGo in manual mode
  tmpNext : BOOL ;	//Global next
  tmpInEnableLN : BOOL ;
  tmpInEnableHN : BOOL ;
  tmpLocalFault : BOOL ;
  tmpLocal : BOOL ;
END_VAR
BEGIN
NETWORK
TITLE =  Start Global
      L     34;
      T     #tmpLenDyn;	//--> Len dynamic data in byte
NETWORK
TITLE = PC Control
//=== Test Object number =====================
      L     "SYS_DirectCtrlDB".PC.ObjectNo;	//PCControl.ObjectNo
      L     #Par.ParObjectNo;	//Input ObjectNo
      <>I;
      JC    aEnd;
//===     Test OType      ========================
      L     1013;	//Input object type
      L     "SYS_DirectCtrlDB".PC.ObjectType;	//PCControl.ObjectType
      <>I;
      JC    aEnd;
//===     Test Handshake =========================
      A     "SYS_DirectCtrlDB".PC.Hsk.FExamine;	// Handshake.FExamine
      JC    aExa;
      A     "SYS_DirectCtrlDB".PC.Hsk.FDefineCmd;	// Handshake.FDefineCmd
      JC    aCmd;
      A     "SYS_DirectCtrlDB".PC.Hsk.FDefinePara;	// Handshake.FDefinePara
      JC    aPar;
aIni: L     2;	// FcInit
      UC    "SYS_DirectCtrl";
      JU    aEnd;
// Write Parameter
aPar: LAR1  P#DBX 58.0;
      L     P##Par;
      L     DW#16#FFFFF;
      AD;
      +AR1;
      L     DBW [AR1,P#8.0];
      T     #Par.ParMonTime;
      L     DBW [AR1,P#10.0];
      T     #Par.ParPulseTimeHN;
      L     DBW [AR1,P#12.0];
      T     #Par.ParPulseTimeLN;
      L     DBW [AR1,P#14.0];
      T     #Par.ParIdlingTime;
      L     DBW [AR1,P#16.0];
      T     #Par.ParDelayTime;
// Write new commands from PC to Interface object
aCmd: A     "SYS_DirectCtrlDB".PC.Cmd1[8];	// CmdLN
      AN    "GCS7_Gr_OutManualOff";	//Global.OutManualOff  [2.10]
      S     #CmdLN;
      A     "SYS_DirectCtrlDB".PC.Cmd1[9];	// CmdHN
      AN    "GCS7_Gr_OutManualOff";	//Global.OutManualOff  [2.10]
      S     #CmdHN;
      A     "SYS_DirectCtrlDB".PC.Cmd1[10];	// CmdNext
      S     #CmdNext;
      A     "SYS_DirectCtrlDB".PC.Cmd1[11];	// CmdFaultReset
      S     #CmdFaultReset;
      A     "SYS_DirectCtrlDB".PC.Cmd1[13];	// CmdManualOn
      S     #InManual;
      A     "SYS_DirectCtrlDB".PC.Cmd1[14];	// CmdReportOn
      S     #InReport;
      A     "SYS_DirectCtrlDB".PC.Cmd2[13];	// CmdManualOff
      R     #InManual;
      A     "SYS_DirectCtrlDB".PC.Cmd2[14];	// CmdReportOff
      R     #InReport;
      AN    "SYS_DirectCtrlDB".PC.Cmd1[1];	// CmdOnTick
      O     "GCS7_Gr_OutManualOff";	//Global.OutManualOff
      JC    aIni;
      L     "SYS_DirectCtrlDB".PC.Cmd3;	// "SYS_PCControl".PC.Cmd3
      T     #Par.InOutManPulseLen;
      JU    aIni;
aExa: TAR2;	// Address Dynamic datas
      T     "SYS_DirectCtrlDB".GC.InDynAddr;	// -->PCControl.GC.InDynAddr
      L     #tmpLenDyn;	// Length Dynamic datas
      T     "SYS_DirectCtrlDB".GC.InDynLen;	// -->PCControl.GC.InDynLen
      L     0;
      T     "SYS_DirectCtrlDB".GC.InParaAddr;	// -->PCControl.GC.InParaAddr
      T     "SYS_DirectCtrlDB".GC.InParaLen;	// -->PCControl.GC.InParaLen
      L     1;	// Code FcExamine
      UC    "SYS_DirectCtrl";
      L     10;	//Revision
      T     "SYS_DirectCtrlDB".GC.Revision;
aEnd: NOP   0;
NETWORK
TITLE =  All State Init
//===Clear tmp Variable
      CLR;
      =     #tmpDelayClear;
      =     #tmpMonClear;
      =     #tmpMonFault;
//Minimum monitoring time                                 
      L     #Par.ParMonTime;	//[2.8]
      L     3;	//[2.8
      >=I;	//[2.8
      JC    ini0;	//[2.8
      T     #Par.ParMonTime;	//[2.8
//===Global Group Orders===
ini0: A     "GCS7_Gr_OutManualOn";	//Gr.OutManualOn
      S     #InManual;
      A     "GCS7_Gr_OutManualOff";	//Gr.OutManualOff
      R     #InManual;
      A     #InManual;
      S     "GCS7_Gr_InManual";	//Gr.InManualMode
      A     #InLocal;
      AN    #InManual;
      =     #tmpLocalFault;	//[4.0]
      A     #tmpLocalFault;	//[4.0]
      O     #InHWStop;	//[4.0]
      O     #InDPFault;	//[4.0]
      =     #tmpLocal;
//---Report is on---
      O     "GCS7_Gr_OutReportAll";	//Gr.OutReportAll
      O     #InReport;
      =     #tmpReport;
NETWORK
TITLE = Start as Pulse
      ON    #InManual;
      O     #CmdLN;
      JC    STP1;
      L     0;
      L     #Par.InOutManPulseLen;
      >=I;
      JC    STP2;
      S     #CmdHN;
      AN    "GCS7_Gr_OutTick200ms";	// Decrement all 200ms
      JC    STP2;
      +     -2;
      T     #Par.InOutManPulseLen;
      L     0;
      >I;
      JC    STP2;
      S     #CmdLN;
STP1: L     0;
      T     #Par.InOutManPulseLen;
STP2: NOP   0;
NETWORK
TITLE = Global Orders Part.2
//===Global Group Orders===
      A     #InEnableLN;
      =     #tmpInEnableLN;
      A     #InEnableHN;
      =     #tmpInEnableHN;
      AN    #InManual;
      ON    #Par.ParManual;
      JC    inJ1;
      A     #StLN;	//---Manual mode without interlocking
      O     #StCtoLN;
      O     #StFault;
      O     #CmdLN;
      AN    #CmdHN;
      =     #tmpInEnableLN;
      A     #StHN;
      O     #StCtoHN;
      O     #CmdHN;
      AN    #CmdLN;	// [2.5]
      =     #tmpInEnableHN;
//---Enable---
inJ1: A     #tmpInEnableLN;	//---Global enable
      X     #tmpInEnableHN;
      =     #tmpEnable;
//---Next---
      O     #CmdNext;	//---automatic StCtoHN
      =     #tmpNext;
//---Input ok---
      A(;
      A     #StLN;	//---Check Input: LN
      A     #InpLN;
      AN    #InpHN;
      O;
      A     #StHN;	// HN
      A     #InpHN;
      AN    #InpLN;
      O;
      AN    #StLN;	//[4.5]
      AN    #StHN;	//[4.5]
      );
      AN    #InpFaultDev;	//[4.0]
      =     #tmpInpOk;
//---Manual StopAndGo---
      A     #CmdLN;
      A     #CmdHN;
      =     #tmpManStopGo;
NETWORK
TITLE = ParDelayTime [4.5]
      NOP   0;
//[4.5]--->
      AN    #tmpInpOk;
      AN    #tmpLocal;	//===No monitoring in local mode
      JC    DTJO;
//--Stop Delay Time Fault ---
      R     #OutDelayFault;
      R     #tmpDelayOver;
      L     #Par.ParDelayTime;
      T     #Par.OutDelayTime;
      JU    DTD9;
//--Run Delay Time Fault ---
DTJO: L     0;
      L     #Par.OutDelayTime;
      >=I;
      ON    "GCS7_Gr_OutTick200ms";	// Decrement all 200ms
      JC    DTD2;
      +     -2;
      T     #Par.OutDelayTime;
DTD2: L     0;
      <=I;
      =     #tmpDelayOver;
      >I;
      =     #OutDelayFault;
DTD9: NOP   0;
//<---[4.5]
NETWORK
TITLE = Monitoring
// Monitoring active only in states StCtoLN and StCtoHN.
// Every transition into these both states will refresh the monitoring time.
      A     #tmpLocal;	//===No monitoring in local mode
      JC    STAT;
//===Condition for not monitoring
      A     #StCtoLN;
      O     #StCtoHN;
      ON    #OutMonFault;	// Clear monitoring information
      JC    MON2;
      R     #OutMonFault;
      S     #tmpMonClear;	// Reset actual value of timer
MON2: AN    #OutMonFault;	//---Condition for monitoring
      JC    STAT;
      A     #InpLN;	// [4.3]
      O     #InpHN;	// [4.3]
      A     #InStopCTime;
      ON    "GCS7_Gr_OutTick200ms";	// Global Tick 200ms
      L     #Par.OutMonTime;
      JC    MO21;
      +     -2;	// Decrement all 200ms
      T     #Par.OutMonTime;
MO21: L     0;
      <=I;	// Check t4/t5 over
      R     #OutMonFault;	// Reset monitoring bits
      =     #tmpMonFault;	//---Condition for monitoring fault
NETWORK
TITLE = States
STAT: A     #StLN;	//===State machine===
      JC    LN;
      A     #StCtoHN;
      JC    CHN;
      A     #StHN;
      JC    HN;
      A     #StCtoLN;
      JC    CLN;
      A     #StNoPosition;
      JC    NPS;
      A     #StFault;
      JC    FLT;
//---Initialise if no state
      S     #StNoPosition;	//[4.4]
      JU    NPS;	//[4.4]  
NETWORK
TITLE = StLN
LN:   AN    #tmpLocal;	//---Condition for StNoPosition: local
      JC    LN1;
      A     #InHWStop;	//[4.0]
      O     #InDPFault;	//[4.0]
      JC    SAVE;	//[4.0]
      AN    #InpLN;
      O;	// [2.6]
      A     #InpLN;	// [2.6]
      A     #InpHN;	// [2.6]
      JC    TNPS;
      JU    SAVE;
LN1:  A     #Par.ParManualFlap;	//===Manual flap function
      AN    #tmpInpOk;	//  without checking t4
      A(;
      AN    #tmpEnable;	// in automatic mode check Enable
      AN    #InManual;
      O;
      A     #InManual;	// not in manual mode
      );
      JC    TCHN;
      A     #tmpDelayOver;	//[4.5] Condition for fault
      JC    LN9;
//===Pulse Valve and Manual Flap
      A     #Par.ParContValve;
      JC    LN3;
      A     #tmpNext;
      AN    #InManual;
      O     #CmdHN;
      A     #tmpInEnableHN;
      AN    #tmpInEnableLN;
      JC    TCHN;
      JU    SAVE;
//===Continuous Valve: automatic StCtoHN
LN3:  A     #tmpNext;
      AN    #InManual;
      AN    #InSeqStop;
      O     #CmdHN;
      A     #tmpInEnableHN;
      JC    TCHN;
      JU    SAVE;
LN9:  R     #StLN;	//---Transition -> StFault
      L     B#(1, 10);	// MessageClass Error fault device
      A     #InpFaultDev;
      JC    xxS4;
      L     B#(1, 11);	// MessageClass Error fault LN
      JU    xxS4;
NETWORK
TITLE = StCtoHN
//---Change into local mode
CHN:  AN    #tmpLocal;
      JC    CHN1;
      A     #InpLN;	// StLN
      AN    #InpHN;
      JC    TLN;
      A     #InpHN;	// StHN
      AN    #InpLN;
      JC    THN;
      JU    TNPS;	// NoPosition
//---Condition for StFault
CHN1: O     #tmpMonFault;
      O     #tmpDelayOver;	//[4.5]
      JC    CHN9;
//---Condition for Pulse Time: not local
      AN    #InpHN;
      O;
      A     #InpLN;
      A     #InpHN;
      JCN   CHD1;
      L     #Par.ParPulseTimeHN;	//[4.5]
      T     #Par.OutTransitionTime;	//[4.5]
      JU    CHN2;	//[4.5]
CHD1: AN    "GCS7_Gr_OutTick200ms";	// Decrement all 200ms
      L     #Par.OutTransitionTime;
      JC    CHD2;
      +     -2;
      T     #Par.OutTransitionTime;
CHD2: L     0;	// Condition for StHN;
      <=I;
      JC    THN;
CHN2: A     #Par.ParContValve;	//---Pulse time (t1) not over
      JC    CHN3;	//===Pulse Valve and Manual Flap
      A     #Par.ParManualFlap;	// Manual flap function
      A     #InpLN;	//  Input changes
      AN    #InpHN;
      AN    #tmpEnable;
      JC    TCLN;
//---Automatic/manual mode: -> StCtoLN
      A     #tmpNext;
      AN    #InManual;
      O     #CmdLN;
      A     #tmpInEnableLN;
      AN    #tmpInEnableHN;
      JC    TCLN;
      A     #Par.ParManualFlap;	// No StopAndGo with ManualFlap
      JC    SAVE;
      AN    #tmpEnable;	// StopAndGo -> StHN
      O     #tmpManStopGo;	// 2.4: CmdLN and CmdHN
      A     #InpHN;
      AN    #InpLN;
      JC    THN;
      AN    #tmpEnable;	// StopAndGo -> StLN
      O     #tmpManStopGo;	// 2.4: CmdLN and CmdHN
      A     #InpLN;
      AN    #InpHN;
      JC    TLN;
      AN    #tmpEnable;	// StopAndGo -> StNoPosition
      O     #tmpManStopGo;	// 2.4: CmdLN and CmdHN
      JC    TNPS;
      JU    SAVE;	// Condition for StCtoHN
//===Continuous Valve:manual StCtoLN      
CHN3: A     #InManual;	//---Manual mode: StCtoLN
      A     #CmdLN;
      ON    #tmpInEnableHN;	//2C:---Automatic + interlocked manual mode: StCtoLN
      O;
      A     #InSeqStop;	// idling activated?
      AN    #InManual;
      JC    TCLN;
      JU    SAVE;
//---Transition -> StFault
CHN9: R     #StCtoHN;
      L     B#(1, 10);	// MessageClass Error fault device
      A     #InpFaultDev;
      JC    xxS4;
      L     B#(1, 12);	// MessageClass Error fault LN      //[4.2]
      A     #InpLN;
      JC    xxS4;
      L     B#(1, 13);	// MessageClass Error fault no position
      JU    xxS4;
NETWORK
TITLE = StHN
HN:   AN    #tmpLocal;	//---Condition for StNoPosition: local
      JC    HN1;
      A     #InHWStop;
      O     #InDPFault;
      AN    #Par.ParContValve;
      JC    SAVE;
      AN    #InpHN;
      O;	// [2.6]
      A     #InpLN;	// [2.6]
      A     #InpHN;	// [2.6]
      JC    TNPS;
      JU    SAVE;
HN1:  A     #Par.ParManualFlap;	//===Hand manual flap function
      AN    #tmpInpOk;	//  without checking t4
      A(;
      AN    #tmpEnable;	// in automatic mode check Enable
      AN    #InManual;
      O;
      A     #InManual;	// not in manual mode
      );
      JC    TCLN;
      A     #tmpDelayOver;	//[4.5] Condition for fault
      JC    HN9;
//===Pulse Valve and Manual Flap
      A     #Par.ParContValve;	//---Input HN ok
      JC    HN3;
      A     #tmpNext;	//---automatic StCtoLN
      O     #CmdLN;
      A     #tmpInEnableLN;
      AN    #tmpInEnableHN;
      O;
      A     #InManual;	//---manual StCtoLN, only with Pulse Valve
      A     #CmdLN;
      AN    #tmpEnable;
      A     #Par.ParPulseValve;
      JC    TCLN;
      JU    SAVE;
//===Continuous Valve: manual StCtoLN
HN3:  A     #InManual;	//---Manual mode: StCtoLN
      A     #CmdLN;
      ON    #tmpInEnableHN;	//2C:---Automatic + interlocked manual mode: StCtoLN
      JC    TCLN;
      O     #InSeqStop;	//---Idling time  
      ON    #OutIdling;	// Condition to reset Idling-Time
      JC    HNI1;
      R     #OutIdling;
      JU    SAVE;
HNI1: ON    #InSeqStop;	// Idling time active ?
      O     #InManual;
      JC    SAVE;
      A     #OutIdling;
      JC    HNI2;
      S     #OutIdling;	// Preset Idling Time
      L     #Par.ParIdlingTime;
      T     #Par.OutTransitionTime;
HNI2: AN    "GCS7_Gr_OutTick200ms";	// Set Idling Time
      L     #Par.OutTransitionTime;
      JC    HNI3;
      +     -2;
      T     #Par.OutTransitionTime;
HNI3: L     0;
      <=I;	// Idling time over
      JC    TCLN;
      JU    SAVE;
HN9:  R     #StHN;	//---Transition -> StFault
      L     B#(1, 10);	// MessageClass Error fault device
      A     #InpFaultDev;
      JC    xxS4;
      L     B#(1, 12);	// MessageClass Error fault HN
      JU    xxS4;
NETWORK
TITLE = StCtoLN
//---Change into local mode ---
CLN:  AN    #tmpLocal;
      JC    CLN1;
      A     #InpLN;	// StLN
      AN    #InpHN;
      JC    TLN;
      A     #InpHN;	// StHN
      AN    #InpLN;
      JC    THN;
      JU    TNPS;	//--> StNoPosition
//---Condition for StFault
CLN1: O     #tmpMonFault;
      O     #tmpDelayOver;	//[4.5]
      JC    CLN9;
//---Condition for Pulse Time: not local---
      AN    #InpLN;
      O;
      A     #InpLN;
      A     #InpHN;
      JCN   CLD1;	//[4.5]
      L     #Par.ParPulseTimeLN;	//[4.5]
      T     #Par.OutTransitionTime;	//[4.5]
      JU    CLN2;
CLD1: AN    "GCS7_Gr_OutTick200ms";	// Decrement all 1s
      L     #Par.OutTransitionTime;
      JC    CLD2;
      +     -2;
      T     #Par.OutTransitionTime;
CLD2: L     0;	// Condition for StLN;
      <=I;
      JC    TLN;
CLN2: A     #Par.ParContValve;	//---Pulse time (t1) not over
      JC    CLN3;	//===Pulse Valve and Manual Flap
      A     #Par.ParManualFlap;	// Manual flap function
      A     #InpHN;	//  Input changes
      AN    #InpLN;
      AN    #tmpEnable;
      JC    TCHN;
      A     #tmpNext;	//-> StCtoHN
      AN    #InManual;
      O     #CmdHN;	//2.4: CmdLN -> CmdHN
      A     #tmpInEnableHN;
      AN    #tmpInEnableLN;
      JC    TCHN;
      A     #Par.ParManualFlap;	// No StopAndGo with ManualFlap
      JC    SAVE;
      AN    #tmpEnable;	//---StopAndGo: automatic StHN
      O     #tmpManStopGo;	// 2.4: CmdLN and CmdHN
      A     #InpHN;
      AN    #InpLN;
      JC    THN;
      AN    #tmpEnable;	// StopAndGo -> StLN
      O     #tmpManStopGo;	// 2.4: CmdLN and CmdHN
      A     #InpLN;
      AN    #InpHN;
      JC    TLN;
      AN    #tmpEnable;	// StopAndGo -> StNoPosition
      O     #tmpManStopGo;	// 2.4: CmdLN and CmdHN
      JC    TNPS;
      JU    SAVE;
//                                ===Continuous Valve
CLN3: A     #tmpNext;	//---automatic StCtoHN
      AN    #InManual;
      AN    #InSeqStop;
      O     #CmdHN;
      A     #tmpInEnableHN;
      JC    TCHN;
      JU    SAVE;
CLN9: R     #StCtoLN;	//---Transition -> StFault
      L     B#(1, 10);	// MessageClass Error fault device
      A     #InpFaultDev;
      JC    xxS4;
      L     B#(1, 11);	// MessageClass Error fault LN //[4.2]
      A     #InpHN;
      JC    xxS4;
      L     B#(1, 13);	// MessageClass Error fault no position
      JU    xxS4;
NETWORK
TITLE =  StNoPosition;
//Valid state for all valves in local mode
//  and in not local mode only for pulse valve and manual flap
NPS:  A     #InpLN;	// -> StLN
      AN    #InpHN;
      JC    TLN;
      A     #InpHN;	// -> StHN
      AN    #InpLN;
      JC    THN;
      A     #tmpLocal;
      JC    SAVE;
//===Manual and automatic mode: InpLN -> StCtoLN
      A     #tmpDelayOver;	//--Condition for StFault
      JC    NPS9;
      A     #Par.ParManualFlap;	//--Condition for StFault
      JC    NPSn;
      A     #tmpNext;	// -> StCtoHN
      AN    #InManual;
      O     #CmdHN;
      A     #tmpInEnableHN;
      AN    #tmpInEnableLN;
      JC    TCHN;
      A     #tmpNext;	// -> StCtoLN
      AN    #InManual;
      O     #CmdLN;
      A     #tmpInEnableLN;
      AN    #tmpInEnableHN;
      JC    TCLN;
      JU    SAVE;
NPS9: R     #StNoPosition;	//---Transition -> StFault
      L     B#(1, 10);	//MessageClass Error fault device
      JU    xxS4;
NPSn: R     #StNoPosition;	//---Transition -> StFault
      L     B#(1, 13);	//MessageClass Error fault no position
      JU    xxS4;
NETWORK
TITLE =  StFault
//Change state conditions
//-----------------------
//All valves:
//FaultReset -> InLocal     -> InpHN  --> StHN
//                             InpLN  --> StLN
//                             no Inp --> StNoPosition
//                             InpHN and InpLN --> StNoPosition
//           -> not InLocal -> InpHN and InpLN --> StFault (reLOG fault)
//
//Pulse valve and Manual flap:
//FaultReset -> not InLocal -> InpHN  --> StCtoHN (start monitoring)
//                             InpLN  --> StCtoLN (  "        "    )
//                             no Inp --> StNoPosition
//Continuous valve:
//FaultReset -> not InLocal -> InpHN  --> StFault (reLOG fault)
//                             InpLN  --> StCtoLN (start monitoring)
//                             no Inp --> StFault (reLOG fault)
xxS4: SET;
      S     #StFault;
      S     "GCS7_Gr_InFaultFlag";	// InFaultFlag
      S     #tmpMonClear;
      T     #tmpLOGvalue;	//[4.1]
      CALL  "SYS_Horn_Code" (
           FcCode                   := 1,
           ParObjectType            := 1013,
           ParObjectNo              := #Par.ParObjectNo,
           ParHornCode              := #Par.ParHornCode);
      L     #tmpLOGvalue;	//[4.1]
      JU    LOG;
//Logic
//Local
FLT:  AN    #tmpLocalFault;
      JC    FLT1;
      A     #InpHN;	// -> StHN
      AN    #InpLN;
      JC    FLT7;
      A     #InpLN;	// -> StLN
      AN    #InpHN;
      JC    FLT6;
      JU    FLT8;	// No Input -> StNoPosition
//Remote
FLT1: AN    #CmdFaultReset;	//---Condition for StFault
      AN    "GCS7_Gr_OutFaultReset";	// OutFaultReset
      JC    SAVE;
      A     #InpFaultDev;	//---Condition for StFault with LOG
      L     B#(1, 10);	// MessageClass Error fault device
      JC    LOG;
      A     #InpLN;	//===All valves: Both Inputs -> StFault
      A     #InpHN;
      L     B#(1, 13);	// MessageClass Error fault no position
      JC    LOG;
      A     #InpLN;	// Input LN -> StCtoLN
      JC    FLT4;
      A     #Par.ParContValve;
      JC    FLT2;	//---Pulse Valve and Manual Flap: not local
      A     #InpHN;	// -> StCtoHN
      JC    FLT5;
      JU    FLT8;	// No Input -> StNoPosition
FLT2: A     #InpHN;	//---Continuous valve
      L     B#(1, 11);	// MessageClass Error fault LN
      JC    LOG;
      L     B#(1, 13);	// MessageClass Error fault no position
      JU    LOG;
FLT4: S     #StCtoLN;	//---Transition -> StCtoLN
      S     #OutMonFault;	// Activate monitoring
      L     #Par.ParPulseTimeLN;
      T     #Par.OutTransitionTime;
      L     #Par.ParMonTime;
      T     #Par.OutMonTime;
      JU    FLM;
FLT5: S     #StCtoHN;	//---Transition -> StCtoHN
      S     #OutMonFault;	// Activate monitoring
      L     #Par.ParPulseTimeHN;
      T     #Par.OutTransitionTime;
      L     #Par.ParMonTime;
      T     #Par.OutMonTime;
      JU    FLM;
FLT6: S     #StLN;	//---Transition -> StLN
      JU    FLM;
FLT7: S     #StHN;	//---Transition -> StHN
      JU    FLM;
FLT8: S     #StNoPosition;	//---Transition -> StNoPosition
FLM:  R     #StFault;
      L     B#(3, 9);	// MessageClass Operate fault cancelled
      JU    LOG;
NETWORK
TITLE = General Transitions
TCLN: SET;	// set VKE=1
      R     #StHN;	//---Transition -> StCtoLN
      R     #StCtoHN;
      R     #StNoPosition;
      S     #StCtoLN;
      R     #OutIdling;
      S     #OutMonFault;	// Activate monitoring
      L     #Par.ParPulseTimeLN;	//[4.5]
      T     #Par.OutTransitionTime;	//[4.5]
      L     #Par.ParMonTime;
      T     #Par.OutMonTime;
      JU    SAVE;
TCHN: SET;	// set VKE=1
      R     #StLN;	//---Transition -> StCtoHN
      R     #StCtoLN;
      R     #StNoPosition;
      S     #StCtoHN;
      S     #OutMonFault;	// Activate monitoring
      L     #Par.ParPulseTimeHN;	//[4.5]
      T     #Par.OutTransitionTime;	//[4.5]
      L     #Par.ParMonTime;
      T     #Par.OutMonTime;
      JU    SAVE;
TLN:  SET;	// set VKE=1
      R     #StCtoHN;	//---Transition -> StLN
      R     #StCtoLN;
      R     #StNoPosition;
      S     #StLN;
      S     #tmpMonClear;
      AN    #tmpReport;	// ReportAll?
      JC    SAVE;
      L     B#(4, 0);	// MessageClass Info LN
      JU    LOG;
THN:  SET;	// set VKE=1
      R     #StCtoHN;	//---Transition -> StHN
      R     #StCtoLN;
      R     #StNoPosition;
      S     #StHN;
      S     #tmpMonClear;
      AN    #tmpReport;	// ReportAll?
      JC    SAVE;
      L     B#(4, 2);	// MessageClass Info HN
      JU    LOG;
TNPS: SET;	// set VKE=1
      R     #StLN;	//---Transition -> StNoPosition
      R     #StCtoHN;
      R     #StHN;
      R     #StCtoLN;
      S     #StNoPosition;
      S     #tmpMonClear;
      JU    SAVE;
NETWORK
TITLE = LOG Message
LOG:  A     #Par.ParLogOff;	//---Set LOG Message
      JC    SAVE;
      T     #tmpLOGvalue;
      L     W#16#FF;
      AW;
      T     #OutAlarmNrLog;
      CALL  "GCS7_LogConvert" (
           ObjectNo                 := #Par.ParObjectNo,
           MsgType                  := #Par.ParMsgType,
           ClassMsgTxt              := #tmpLOGvalue,
           OType                    := 1013);	// LOG Message Converter / Entry / Contains Class and TextNo
NETWORK
TITLE = Global End
SAVE: CLR;	//---Clear all commands
      =     #CmdLN;
      =     #CmdHN;
      =     #CmdNext;
      =     #CmdFaultReset;
      A     #StCtoHN;	//---Condition for setting Output HN
      AN    #Par.ParManualFlap;
      O;
      A     #StHN;
      A     #Par.ParContValve;
      AN    #tmpLocal;
      =     #OutpHN;
      A     #StCtoLN;	//---Condition for setting Output LN
      A     #Par.ParPulseValve;
      =     #OutpLN;
//--Output for group 
      AN    #InLocal;
      O     #InManual;
      A     #InDPFault;
      S     "GCS7_Gr_InDPFault";
      AN    #InLocal;
      O     #InManual;
      A     #InHWStop;
      S     "GCS7_Gr_InHWStop";
//---Clear actual value of timer
      AN    #tmpMonClear;
      JC    STC;
      T     #Par.OutMonTime;	// Clear monitoring timer
      R     #OutMonFault;
NETWORK
TITLE = State Code
STC:  A     #StFault;
      JC    STC8;	//Code: Fault
//--------------------
      AN    #StLN;
      JC    STC2;
      L     41;	//Code: StLN.HWStop
      A     #InHWStop;
      JC    STC9;
      L     51;	//Code: StLN.DPFault
      A     #InDPFault;
      JC    STC9;
      L     1;	//Code: LN
      JU    STC9;
//--------------------
STC2: A     #InStopCTime;	//[4.3]
      A     #StCtoHN;	//[4.3]
      L     12;	//[4.3]
      JC    STC9;
      A     #StCtoHN;
      L     2;	//Code: change to HN
      JC    STC9;
//--------------------
      AN    #StHN;
      JC    STC4;
      L     43;	//Code: StHN.HWStop
      A     #InHWStop;
      JC    STC9;
      L     53;	//Code: StHN.DPFault
      A     #InDPFault;
      JC    STC9;
      L     3;	//Code: HN
      JC    STC9;
//--------------------
STC4: A     #InStopCTime;	//[4.3]
      A     #StCtoLN;	//[4.3]
      L     14;	//[4.3]
      JC    STC9;
      A     #StCtoLN;
      L     4;	//Code: Change to LN
      JC    STC9;
//--------------------
      AN    #StNoPosition;
      JC    STC8;
      L     45;	//Code: StNoPosition.HWStop
      A     #InHWStop;
      JC    STC9;
      L     55;	//Code: StNoPosition.DPFault
      A     #InDPFault;
      JC    STC9;
      L     5;	// Code: StNoPosition
      JU    STC9;
STC8: A     #InpFaultDev;
      L     31;
      JC    STC9;	// StFault.InpFaultDev
      L     32;	// Code: fault
STC9: L     #StCode;	// Old state code
      TAK;
      T     #StCode;	// Save state code
      <>I;
      L     3;	// Load code for CBit methode
      CC    "SYS_CBitCtrl";
END_FUNCTION_BLOCK

FUNCTION_BLOCK "GCS7_E_DigInput"	// FB 14
TITLE = DigInpCont
//
//COPYRIGHT:    (C) 1996  BUHLER AG, CH-9240 UZWIL, SWITZERLAND
//
//PRODUCT:      GCS7
//
//TITLE:        Element Digital Input Continuous
//
//-------------------------------------------------------------------------
//
//IDENT:        AUTHOR:             DEPT:                       DATE:
//FB14.4.7      A. Egli             BASE                        18-Jun-2008
//              Check Sum Par.OutTransitionTime>=0 with SPPZ 
//FB14.4.6      A. Egli             BASE                        19-Mai-2008
//              Check Sum Par.OutTransitionTime>0
//FB14.4.5      A. Egli             CT3                         04-Oct-2007
//              Send OutpFaultReset also if element is not monitoried
//FB14.4.4      A. Egli             CT3                         16-Mai-2006
//              Transition StFalse to StTrue
//FB14.4.3      A. Egli             CT3                         24-Nov-2004
//              Local Mode: No prealarm as long InLocal
//FB14.4.2      A. Egli             CT3                         24-Nov-2003
//              Local Mode: Pulse length OutpFaultReset  = 1s
//FB14.4.1      A. Egli             CT3                         18-Nov-2003
//              Transition StTrue to StFault, when 
//                ParDelayChange=0 and ParDelayFalse=0
//FB14.4.0      A. Egli             CT3                          7-Nov-2002
//              New Release with one block 
//              OutpFaultReset in Local mode (3.5)
//FB14.3.4      A. Egli             CT3                         22-Mai-2002
//              Count par.OutMonTime only if monitoring is active
//FB14.3.3      A. Egli             CT3                         12-Apr-2002
//              Reset CmdFaultReset if no StFaultStFault
//FB14.3.2      A. Egli             CT3                         18-Mar-2002
//              Set OutpFaultReset only in StFault
//FB14.3.1      A. Egli             CT3                         19-Jan-2002
//              Length OutpFaultReset = 1s
//              Timebase 200ms for monitoring function
//FB14.3.0      A. Egli             CT3                         29-Okt-2001
//              StCode 30: InpFaultDev=1 and InLocal=1              
//              StCode 31: InpFaultDev=1 and InLocal=0              
//              StCode 11: StFalse.Warning  , StCode 13: StTrue.Warning           
//              StCode 12: StCtoTrue.Warning, StCode 14: StCtoFalse.Warning       
//FB14.2.10     A. Egli             CT3                         29-Okt-2001
//              InLocal: StFault-->StTrue; StFault-->StFalse;
//FB14.2.9      A. Egli             CT3                         04-Okt-2001
//              1 working Condition:  
//                No monitoring fault during StCToTrue or StCToFalse
//FB14.2.8      A. Egli             CT3                         21-Jun-2000
//              Detect immediately change from InMonTrue to InMonFalse
//FB14.2.7      A. Egli             CT3                          2-Mai-2000
//              - Restart monitoring time only with positv edge InMonXxxx
//              - Transition StCtoTrue --> StFalse without hysteresis           
//              - Transition StCtoFalse--> StTrue  without hysteresis
//              - Length OutpFaultReset = 500ms
//              - CmdRunTimeoutTime
//FB14.2.6      S. Kalberer         CT3                         26-Jan-2000
//              2-WorkCond.: run out monitoring time
//FB14.2.5      S. Kalberer         CT3                         11-Jan-2000
//              2-WorkCond.: No hysteresis anymore           
//FB14.2.4      S. Kalberer         CT3                         02-Nov-1999
//              2-WorkCond.: No restart of monitoring time
//FB14.2D       A. Egli             CT3                         11-Jan-1999
//              PC Direct Control: Init is code 2 not 4
//FB14.2C       A. Egli             CT3                          5-Jan-1999
//              OutFlagPos, OutFlagNeg, OutTrue
//FB14.2B       A. Egli             CT3                          5-Jan-1999
//              OutpFaultReset
//FB14.2A       A. Egli             CT3                         04-Mai-1998
//              StFault = StCode 32
//FB14.1A       S. Kalberer         AEE61                       11-Jul-1997
//              1st Release in S7
//
//-------------------------------------------------------------------------
//
//PURPOSE:      MANUAL : see [DICxxMAN]
//
//RESTRICTIONS: S7
//              ACCU2: Pointer to dynamic datas of the element
//              ACCU1: Pointer to parameter datas of the element
//
//-------------------------------------------------------------------------
//=======================================================
//Log Message: 
//------------------------------------------------------
// 0  false
// 2  true
// 9  fault cancelled
//10  fault device
//11  fault true
//12  fault false
//13  prealarm true
//14  prealarm false
//
//=======================================================
//StCode:  State               
//------------------------------------------------------
//32  StFault                  StFault+InpFaultDev=0 
//31  StFault.DEV              StFault+InpFaultDev=1 
// 1  StFalse               
//11  StFalse.Warning          StFalse+OutWarning
//41  StFalse.HWStop           StFalse+HWStop 
//51  StFalse.DPFault          StFalse+DPFault
//61  StFalse.FaultDev         InLocal=1 +InpFaultDef +InpTrue=0
// 2  StCtoTrue             
//12  StCtoTrue.Warning     
// 3  StTrue                
//13  StTrue.Warning           StTrue+OutWarning
//43  StTrue.HWStop            StTrue+InHWStop
//53  StTrue.DPFault           StTrue+InDPFault
//63  StTrue.FaultDev          InLocal=1 +InpFaultDef +InpTrue=1
// 4  StCtoFalse             
//14  StCtoFalse.Warning       StCtoFalse+OutWarning
//
//
//
AUTHOR : EA
FAMILY : GCS7LL
NAME : DIC
VERSION : 4.7
VAR
  StCode : INT ;	//Element state code
  InMonTrue : BOOL ;	//After t4 must be StTrue, otherwise it is a process fault
  InMonFalse : BOOL ;	//After t5 must be StFalse, otherwise it is a process fault
  InPreAlarmTrue : BOOL ;	//LOG Pre-alarm if state is not StTrue
  InPreAlarmFalse : BOOL ;	//LOG Pre-alarm if state is not StFalse
  InStopTrueTime : BOOL ;	//Stop delay time t2
  InStopFalseTime : BOOL ;	//Stop delay time t3
  InpTrue : BOOL ;	//Digital input: signal 'True'; target state is StTrue
  InpFaultDev : BOOL ;	//Digital input: fault device
  CmdRstTrueTime : BOOL ;	//Restart delay time changing from StFalse to StTrue (t2)
  CmdRstFalseTime : BOOL ;	//Restart delay time changing from StTrue to StFalse (t3)
  CmdRunTimeoutTime : BOOL ;	//Run timeout time (only 1 working condition)
  CmdFaultReset : BOOL ;	//Command to reset fault
  InLocal : BOOL ;	//1= Local mode (automatic fault reset)
  spare0305 : BOOL ;	//Copy of InMonTrue to detect change form InMonTrue to InMonFalse
  InReport : BOOL ;	//Report of all state transitions
  OutTimeoutTime : BOOL ;	//Timeout time 1 working condition active
  InHWStop : BOOL ;	//HW stop is detected, no fault
  InDPFault : BOOL ;	//DP-Fault is detected, no fault
  OutPreAlarmTrue : BOOL ;	//Flag PreAlarmTrue is done
  OutPreAlarmFalse : BOOL ;	//Flag PreAlarmFalse is done
  OutFlagPos : BOOL ;	//Positive flag InpTrue
  OutFlagNeg : BOOL ;	//Negative flag InpTrue
  OutpFaultReset : BOOL ;	//Reset alarm
  OutTrue : BOOL ;	//Copy of input signal
  StFalse : BOOL ;	//Signal is 'False', delay time finished, monitoring is off
  StCtoTrue : BOOL ;	//Changing to 'True', signal is 'True'
  StTrue : BOOL ;	//Signal is 'True', delay time finished
  StCtoFalse : BOOL ;	//Changing to 'False', signal is 'False'
  StFault : BOOL ;	//Signal has not requested value, monitoring is active
  OutAlarmNrLog : INT ;	//Last textnumber send to log
  Par : STRUCT
   ParObjectNo : INT ;	//Is used for communication with PC, e.g. for message
   ParMsgType : INT ;	//Is used for message (translation of state)
   ParHornCode : INT ;	//Is used by horn module
   ParLogOff : BOOL ;	//Report is off
   spare0401 : BOOL ;
   Par2WorkingCond : BOOL ;	//Element has 2 defined working conditions
   ParFaultRetry : BOOL ;	//Retry after fault with monitoring- and delay-time
   ParBinLevel : BOOL ;	//Hold old state, if HWStop of DPFault
   ParDelayChange : INT ;	//Delay time, if the input changes, until the element changes its state
   ParDelayTrue : INT ;	//Time to change from StFalse to StTrue
   ParDelayFalse : INT ;	//Time to change from StTrue to StFalse
   ParTimeoutTrue : INT ;	//If InMonTrue: after this time state has to be 'StTrue', otherwise StFault
   ParTimeoutFalse : INT ;	//If InMonFalse: after this time state has to be 'StFalse', otherwise StFault
   OutMonTime : INT ;	//Actual time: monitoring
   OutTransitionTime : INT ;	//Actual time: changing state
   OutMonTrue : BOOL ;	//Monitoring time true is running
   OutMonFalse : BOOL ;	//Monitoring time false is running
   OutFlagFaultDev : BOOL ;	//Flag InpFaultDev
   OutDelayTime : INT ;	//Actual time: DelayTime
  END_STRUCT ;
END_VAR
VAR_TEMP
  tmpLOGvalue : WORD ;	//LOG value
  tmpAddrPara : DWORD ;	//store the Instance Pointer
  tmpLenDyn : DINT ;
  tmpReport : BOOL ;	//Global LOG all
  tmpMonFault : BOOL ;	//Global monitor fault
  tmpMonOver : BOOL ;	//Monitoring time over
  tmp2WorkingCond : BOOL ;	//Monitoring time over
  tmpOutDelayDone : BOOL ;	//ParDelayTime Done
  tmpLocalFault : BOOL ;
  tmpLocal : BOOL ;
END_VAR
BEGIN
NETWORK
TITLE =  Start Global
      L     32;
      T     #tmpLenDyn;	//--> Len dynamic data in byte
NETWORK
TITLE = PC Control
//=== Test Object number =====================
      L     "SYS_DirectCtrlDB".PC.ObjectNo;	//PCControl.ObjectNo
      L     #Par.ParObjectNo;	//Input ObjectNo
      <>I;
      JC    Ctrl;
//=== Test OType      ========================
      L     1014;	//Input object type
      L     "SYS_DirectCtrlDB".PC.ObjectType;	//PCControl.ObjectType
      <>I;
      JC    Ctrl;
//=== Test Handshake =========================
      A     "SYS_DirectCtrlDB".PC.Hsk.FExamine;	// Handshake.FExamine
      JC    pExa;
      A     "SYS_DirectCtrlDB".PC.Hsk.FDefineCmd;	// Handshake.FDefineCmd
      JC    pCmd;
      A     "SYS_DirectCtrlDB".PC.Hsk.FDefinePara;	// Handshake.FDefinePara
      JC    pPar;
pIni: L     2;	// FcInit  [2D]
      UC    "SYS_DirectCtrl";
      JU    Ctrl;
// Write new commands from PC to Interface object
pPar: LAR1  P#DBX 58.0;
      L     P##Par;
      L     DW#16#FFFFF;
      AD;
      +AR1;
      L     DBW [AR1,P#8.0];
      T     #Par.ParDelayChange;
      L     DBW [AR1,P#10.0];
      T     #Par.ParDelayTrue;
      L     DBW [AR1,P#12.0];
      T     #Par.ParDelayFalse;
      L     DBW [AR1,P#14.0];
      T     #Par.ParTimeoutTrue;
      L     DBW [AR1,P#16.0];
      T     #Par.ParTimeoutFalse;
pCmd: A     "SYS_DirectCtrlDB".PC.Cmd1[2];	// CmdPreAlarmTrueOn
      S     #InPreAlarmTrue;
      A     "SYS_DirectCtrlDB".PC.Cmd1[3];	// CmdPreAlarmFalseOn
      S     #InPreAlarmFalse;
      A     "SYS_DirectCtrlDB".PC.Cmd1[8];	// CmdRstTrueTime
      S     #CmdRstTrueTime;
      A     "SYS_DirectCtrlDB".PC.Cmd1[9];	// CmdRstFalseTime
      S     #CmdRstFalseTime;
      A     "SYS_DirectCtrlDB".PC.Cmd1[11];	// CmdFaultReset
      S     #CmdFaultReset;
      A     "SYS_DirectCtrlDB".PC.Cmd1[12];	// CmdFaultReset
      S     #CmdRunTimeoutTime;
      A     "SYS_DirectCtrlDB".PC.Cmd1[14];	// CmdReportOn
      S     #InReport;
      A     "SYS_DirectCtrlDB".PC.Cmd2[2];	// CmdPreAlarmTrueOff
      R     #InPreAlarmTrue;
      A     "SYS_DirectCtrlDB".PC.Cmd2[3];	// CmdPreAlarmFalseOff
      R     #InPreAlarmFalse;
      A     "SYS_DirectCtrlDB".PC.Cmd2[14];	// CmdReportOff
      R     #InReport;
      JU    pIni;
pExa: TAR2;	// Address Dynamic datas
      T     "SYS_DirectCtrlDB".GC.InDynAddr;	// -->PCControl.GC.InDynAddr
      L     #tmpLenDyn;	// Length Dynamic datas
      T     "SYS_DirectCtrlDB".GC.InDynLen;	// -->PCControl.GC.InDynLen
      L     0;
      T     "SYS_DirectCtrlDB".GC.InParaAddr;	// -->PCControl.GC.InParaAddr
      T     "SYS_DirectCtrlDB".GC.InParaLen;	// -->PCControl.GC.InParaLen
      L     1;	// Code FcExamine
      UC    "SYS_DirectCtrl";
      L     10;	//Revision
      T     "SYS_DirectCtrlDB".GC.Revision;
NETWORK
TITLE =  All State Init
//===Clear tmp Variable, when nessecary
Ctrl: A     "GCS7_Gr_OutFaultReset";	// Gr.OutFaultReset
      S     #CmdFaultReset;
      AN    #InpTrue;
      A     #OutTrue;
      =     #OutFlagNeg;
      A     #InpTrue;
      FP    #OutTrue;
      =     #OutFlagPos;
//Local
      A     #InLocal;
      =     #tmpLocalFault;	//[4.0]
      A     #tmpLocalFault;	//[4.0]
      O     #InHWStop;	//[4.0]
      O     #InDPFault;	//[4.0]
      =     #tmpLocal;
//---Report is on---
      O     "GCS7_Gr_OutReportAll";	//---Gr.OutReportAll
      O     #InReport;
      =     #tmpReport;
      A     #CmdRunTimeoutTime;
      S     #OutTimeoutTime;
      R     #Par.OutMonTrue;
      R     #Par.OutMonFalse;
      A     #Par.Par2WorkingCond;
      O     #OutTimeoutTime;
      =     #tmp2WorkingCond;
NETWORK
TITLE = Monitoring Time 2 working conditions
      AN    #tmp2WorkingCond;
      R     #tmpMonFault;
      R     #Par.OutMonTrue;
      R     #Par.OutMonFalse;
      JC    TiJ0;
//Positiv flag of monitoring function => Start Delay time?
      A     #InMonTrue;
      FP    #Par.OutMonTrue;
      L     #Par.ParTimeoutTrue;
      JC    M021;
      A     #InMonFalse;
      FP    #Par.OutMonFalse;
      O     #CmdRunTimeoutTime;
      L     #Par.ParTimeoutFalse;
      JC    M021;
      JU    M022;
M021: T     #Par.OutMonTime;
M022: L     0;
      L     #Par.OutMonTime;	// Monitoring time over
      >=I;
      ON    "GCS7_Gr_OutTick200ms";	// Gr.OutTick200ms  [3.1]
      O;
      AN    #Par.OutMonTrue;	//[3.4]
      AN    #Par.OutMonFalse;	//[3.4]
      O;	//[3.4]
      A     #CmdRunTimeoutTime;	//[3.4]
      AN    #Par.Par2WorkingCond;	//[3.4]
//      UN    #InMonTrue              //[3.4]
//      UN    #InMonFalse             //[3.4]
//      UN    #OutTimeoutTime         //[3.4]
      L     #Par.OutMonTime;
      JC    MO23;
      +     -2;	// Decrement all 200ms  [3.1]
      T     #Par.OutMonTime;
MO23: L     0;
      <=I;	// Check t4/t5 over
      =     #tmpMonOver;
//---Condition for monitoring fault 
      A     #InMonTrue;
      A     #tmpMonOver;
      AN    #StTrue;
      A(;	//[2.9]
      AN    #StCtoFalse;	//[2.9]
      O     #Par.Par2WorkingCond;	//[2.9]
      );	//[2.9]
      O;
      A     #InMonFalse;
      A     #tmpMonOver;
      AN    #StFalse;
      A(;	//[2.9]
      AN    #StCtoTrue;	//[2.9]
      O     #Par.Par2WorkingCond;	//[2.9]
      );	//[2.9]
      =     #tmpMonFault;
//--- CmdRunTimeout is Done by 1 working condition
      A     #tmpMonOver;
      O     #Par.Par2WorkingCond;
      R     #OutTimeoutTime;
NETWORK
TITLE = TransitionTime
//--- Start DelayTime:
TiJ0: AN    #OutFlagPos;
      JC    TiJ1;
      L     #Par.ParDelayTrue;
      JU    TiJ2;
TiJ1: AN    #OutFlagNeg;
      JC    TiDo;
      L     #Par.ParDelayFalse;
TiJ2: L     #Par.ParDelayChange;
      +I;
      T     #Par.OutTransitionTime;	// Set delay time and bit
      JPZ   TiDo;	//[4.7]
      L     32767;	//[4.6]
      T     #Par.OutTransitionTime;	//[4.6]
//--- Run DelayTime:
TiDo: L     0;	//  and time
      L     #Par.OutTransitionTime;	// Check delay time on zero
      >=I;
      JC    TiT2;
      A     #InStopTrueTime;	//---Stop time: delay monitoring
      A     #InpTrue;
      AN    #StFalse;
      AN    #StTrue;
      O;
      A     #InStopFalseTime;
      AN    #InpTrue;
      AN    #StFalse;
      AN    #StTrue;
      ON    "GCS7_Gr_OutTick200ms";	// Gr.OutTick200ms  [3.1]
      JC    TiT2;
      +     -2;	// Decrement all 200ms  [3.1]
      T     #Par.OutTransitionTime;	// Set DelayTime
TiT2: NOP   0;
NETWORK
TITLE = Delay Time
      A     #StFalse;
      A     #InpTrue;
      O;
      A     #StTrue;
      AN    #InpTrue;
      O;
      A     #InpFaultDev;	//1+2 Working Condition
      JC    DTJ1;
      R     #tmpOutDelayDone;
      L     #Par.ParDelayChange;
      T     #Par.OutDelayTime;
      L     0;	//[4.1]
      >I;	//[4.1]
      JC    DTJ0;	//[4.1]
DTJ1: AN    "GCS7_Gr_OutTick200ms";	// Gr.OutTick200ms  [3.1]
      JC    DTJ2;
      L     #Par.OutDelayTime;
      +     -2;	// Decrement all 200ms  [3.1]
      T     #Par.OutDelayTime;
DTJ2: L     #Par.OutDelayTime;
      L     0;
      <=I;	// Check t4/t5 over
      =     #tmpOutDelayDone;
      JCN   DTJ0;
      T     #Par.OutDelayTime;
DTJ0: NOP   0;
NETWORK
TITLE = States
STAT: A     #StFalse;	//===State machine===
      R     #OutPreAlarmFalse;
      JC    S0;
      A     #StCtoTrue;
      JC    S1R;
      A     #StTrue;
      R     #OutPreAlarmTrue;
      JC    S2;
      A     #StCtoFalse;
      JC    S3A;
      A     #StFault;
      JC    S4T;
//Initialise: goto StFalse or StTrue
      AN    #InpTrue;
      S     #StFalse;
      NOT;
      S     #StTrue;
      JU    STAT;
NETWORK
TITLE = StFalse
//---Condition for StFault 
S0:   A     #InHWStop;	//[4.0]
      O     #InDPFault;	//[4.0]
      A     #Par.ParBinLevel;	//[4.0]
      JC    SAVE;	//[4.0]
      A     #InMonTrue;	//1Working Condition
      AN    #InpTrue;	//1Working Condition
      AN    #tmp2WorkingCond;	//1Working Condition
      O;
      A     #InpFaultDev;	//1+2 Working Condition
      A     #tmpOutDelayDone;	//[4.0]
      O     #tmpMonFault;	//2 Working Condition
      AN    #tmpLocal;
      JC    S0S4;
//---Condition for StTrue
      L     #Par.ParDelayTrue;	//[4.4]
      L     0;	//[4.4]
      ==I;	//[4.4]
      AN    #InMonFalse;	//[4.4]
      A     #InpTrue;	//[4.4]
      R     #StFalse;	//[4.4]
      S     #StTrue;	//[4.4]
      JC    SAVE;	//[4.4]
//---Condition for StFalse
      AN    #InpTrue;	// and InpTrue
      ON    #tmpOutDelayDone;	//[4.0]
      JC    SAVE;
//---Transition -> StCtoTrue
      R     #StFalse;
      S     #StCtoTrue;
      JU    SAVE;
//---Transition -> StFault
S0S4: R     #StFalse;
      JU    xxS4;
NETWORK
TITLE = StCtoTrue
//---Condition for StFalse
S1R:  A     #InHWStop;	//[4.0]
      O     #InDPFault;	//[4.0]
      A     #Par.ParBinLevel;	//[4.0]
      JC    SAVE;	//[4.0]
      AN    #InpTrue;	//2.5, 2.7: No hysteresis
      JC    S1S0;
//---Restart delay time
      AN    #CmdRstTrueTime;
      JC    S1R1;
      L     #Par.ParDelayTrue;
      T     #Par.OutTransitionTime;
//---Condition for StFault : 1 WorkCondition
S1R1: L     #Par.OutTransitionTime;
      L     0;
      <=I;	// Check t2 over
      AN    #tmp2WorkingCond;
      A     #InMonFalse;
      AN    #tmpLocal;
      JC    S1S4;
//---Condition for StFalse
      <=I;	// Check t2 over
      JC    S1S2;	//-->StTrue 
//---Condition for StFault 
      A     #InpFaultDev;	//1+2 Working Condition 
      A     #tmpOutDelayDone;	//[4.0]
      O     #tmpMonFault;	//2 Working Condition
      AN    #tmpLocal;
      JC    S1S4;
      JU    SAVE;
//---Transition -> StTrue
S1S2: R     #StCtoTrue;
      S     #StTrue;
      JU    LOG1;
//---Transition -> StFalse
S1S0: R     #StCtoTrue;
      S     #StFalse;
      JU    LOG1;
//---Transition -> StFault
S1S4: R     #StCtoTrue;
      JU    xxS4;
NETWORK
TITLE = StTrue
//---Condition for StFault 
S2:   A     #InHWStop;	//[4.0]
      O     #InDPFault;	//[4.0]
      A     #Par.ParBinLevel;	//[4.0]
      JC    SAVE;	//[4.0]
      A     #InMonFalse;	//1Working Condition
      A     #InpTrue;	//1Working Condition
      AN    #tmp2WorkingCond;	//1Working Condition
      O;
      A     #InpFaultDev;	//1+2 Working Condition
      A     #tmpOutDelayDone;	//[4.0]
      O     #tmpMonFault;	//2 Working Condition
      AN    #tmpLocal;
      JC    S2S4;
//---Condition for StTrue
      A     #InpTrue;
      ON    #tmpOutDelayDone;	//[4.0]
      JC    SAVE;
//---Condition directly change to StFault //[4.1]
      L     #Par.ParDelayChange;	//[4.1]
      L     0;	//[4.1]
      ==I;	//[4.1]
      A(;	//[4.1]
      L     #Par.ParDelayFalse;	//[4.1]
      ==I;	//[4.1]
      );	//[4.1]
      A     #InMonTrue;	//[4.1]
      AN    #tmp2WorkingCond;	//[4.1]
      AN    #InLocal;	//[4.1]
      JC    S2S4;	//[4.1]
//---Condition for StCtoFalse
      R     #StTrue;	//---Transition -> StCtoFalse
      S     #StCtoFalse;	//---Transition -> StCtoFalse
      JU    SAVE;
S2S4: R     #StTrue;	//---Transition -> StFault
      JU    xxS4;
NETWORK
TITLE = StCtoFalse
//---Condition for StFault , only 2work. condition
//Condition for StTrue
S3A:  A     #InHWStop;	//[4.0]
      O     #InDPFault;	//[4.0]
      A     #Par.ParBinLevel;	//[4.0]
      JC    SAVE;	//[4.0]
      A     #InpTrue;
      JC    S3A7;
//---Restart delay time
      AN    #CmdRstFalseTime;
      JC    S3A1;
      L     #Par.ParDelayFalse;	// Set actual value of timer
      T     #Par.OutTransitionTime;
//---Condition StFault by 1WorkCond
S3A1: L     #Par.OutTransitionTime;
      L     0;
      <=I;	// Check t2 over
      AN    #tmp2WorkingCond;
      A     #InMonTrue;
      AN    #tmpLocal;
      JC    S3S4;
//---Condition StFalse
      <=I;	// Check t2 over
      JC    S3S1;
//---Condition for StFault : 1+2 WorkCondition
      A     #InpFaultDev;
      A     #tmpOutDelayDone;	//[4.0]
      O     #tmpMonFault;
      AN    #tmpLocal;
      JC    S3S4;
      JU    SAVE;
//---Transition -> StFalse
S3S1: R     #StCtoFalse;
      S     #StFalse;
      JU    LOG1;
//2.5:---Transition -> StTrue
S3A7: R     #StCtoFalse;
      S     #StTrue;
      JU    LOG1;
//---Transition -> StFault
S3S4: R     #StCtoFalse;
      JU    xxS4;
NETWORK
TITLE =  StFault
// Any transiton to Fault  
xxS4: SET;
      S     #StFault;
      S     "GCS7_Gr_InFaultFlag";	// Gr.InFaultFlag
      CALL  "SYS_Horn_Code" (
           FcCode                   := 1,
           ParObjectType            := 1014,
           ParObjectNo              := #Par.ParObjectNo,
           ParHornCode              := #Par.ParHornCode);
      JU    LOG4;
//==Logic====
//---Transition -> StCtoTrue            
S4T:  A     #tmpLocalFault;
      A     #InpTrue;
      R     #StFault;
      S     #StTrue;	//[3.10]
      JC    S4M;	//[3.9] SPB S4S1
//---Transition -> StCtoFalse           
      A     #tmpLocalFault;
      R     #StFault;
      S     #StFalse;	//[3.10]
      JC    S4M;	//[3.9] SPB S4S3
      A     #InpFaultDev;
      A     #tmpOutDelayDone;
      AN    #Par.OutFlagFaultDev;	//[4.0]
      JC    LOG4;
//---Condition for StFault retry
      AN    "GCS7_Gr_OutTick1s";	// Gr.OutTick1s [3.1]
      ON    #OutpFaultReset;
      JC    SAVE;
      R     #OutpFaultReset;
// Retry message InpFaultDev
      A     #InpFaultDev;
      JC    LOG4;
// Retry message Monitoring true
      AN    #InMonTrue;
      JC    S4T3;
      A     #InpTrue;
      A     #tmp2WorkingCond;
      JC    S4S2;
      A     #InpTrue;
      JC    S4S1;
      A     #OutTimeoutTime;
      O     #Par.ParFaultRetry;
      A     #tmp2WorkingCond;	//   RetryFault only with 2WorkCondition
      JC    S4S3;
      JU    LOG4;	// by monitoring true
// Retry message Monitoring false
S4T3: AN    #InMonFalse;
      JC    S4T4;
      AN    #InpTrue;	// Input = false
      A     #tmp2WorkingCond;
      JC    S4S0;
      AN    #InpTrue;	// Input = false
      JC    S4S3;
      A     #OutTimeoutTime;
      O     #Par.ParFaultRetry;
      A     #tmp2WorkingCond;	//   RetryFault only with 2WorkCondition
      JC    S4S1;
      JU    LOG4;	// by monitoring false
//---Transition -> StFalse
S4S0: R     #StFault;
      S     #StCtoFalse;
      JU    S4M;
//---Transition -> StTrue
S4S2: R     #StFault;
      S     #StCtoTrue;
      JU    S4M;
// If no monitoring function, transition to StCtoFalse 
S4T4: AN    #InpTrue;
      JC    S4S3;	//-->StCtoFalse
// If no monitoring function, transition to StCtoTrue
//---Transition -> StCtoTrue
S4S1: R     #StFault;
      S     #StCtoTrue;
      JU    S4M;
//---Transition -> StCtoFalse
S4S3: R     #StFault;
      S     #StCtoFalse;
//---Any Transition 
S4M:  A     #Par.ParFaultRetry;	//---Condition for Retrigger monitoring time:
      R     #Par.OutMonTrue;
      R     #Par.OutMonFalse;
      JU    LOG0;	//   without retriggering monitoring time
NETWORK
TITLE = LOG Message
//LOG transition to StFalse/StTrue
LOG1: AN    #tmpReport;	// Report all?
      JC    SAVE;
      A     #StTrue;
      L     B#(4, 2);	// MessageClass Info true
      JC    LOG;
      A     #StFalse;
      L     B#(4, 0);	// MessageClass Info flase
      JC    LOG;
      JC    SAVE;
//LOG transition to fault
LOG4: L     B#(1, 10);	// MessageClass Error fault device
      A     #InpFaultDev;
      =     #Par.OutFlagFaultDev;
      JC    LOG;
      L     B#(1, 12);	// MessageClass Error fault false
      A     #InMonTrue;	// by monitoring true
      JC    LOG;
      L     B#(1, 11);	// MessageClass Error fault true
      JU    LOG;
//Log fault cancelled
LOG0: L     B#(3, 9);	// MessageClass Operate fault cancelled
LOG:  A     #Par.ParLogOff;	//---Set LOG Message
      JC    SAVE;
      T     #tmpLOGvalue;
      L     W#16#FF;
      AW;
      T     #OutAlarmNrLog;
      CALL  "GCS7_LogConvert" (
           ObjectNo                 := #Par.ParObjectNo,
           MsgType                  := #Par.ParMsgType,
           ClassMsgTxt              := #tmpLOGvalue,
           OType                    := 1014);	// LOG Message Converter / Entry / Contains Class and TextNo
NETWORK
TITLE = Global End
//===Check PreAlarm
//---Condition for PreAlarm
SAVE: AN    #InPreAlarmTrue;
      O     #OutPreAlarmTrue;
      O     #StTrue;
      O     #tmpLocal;	//[4.3]
      JC    SAV0;
      S     #OutPreAlarmTrue;
      S     "GCS7_Gr_InFaultFlag";	// Gr.InFaultFlag
      CALL  "SYS_Horn_Code" (
           FcCode                   := 1,
           ParObjectType            := 1014,
           ParObjectNo              := #Par.ParObjectNo,
           ParHornCode              := #Par.ParHornCode);
      L     B#(1, 13);	// MessageClass Error prealarm true
      JU    LOG;
//---Condition for PreAlarm
SAV0: AN    #InPreAlarmFalse;
      O     #OutPreAlarmFalse;
      O     #StFalse;
      O     #tmpLocal;	//[4.3]
      JC    SAV1;
      S     #OutPreAlarmFalse;
      S     "GCS7_Gr_InFaultFlag";	// Gr.InFaultFlag
      CALL  "SYS_Horn_Code" (
           FcCode                   := 1,
           ParObjectType            := 1014,
           ParObjectNo              := #Par.ParObjectNo,
           ParHornCode              := #Par.ParHornCode);
      L     B#(1, 14);	// MessageClass Error prealarm false
      JU    LOG;
//===Clear all commands
SAV1: CLR;
      =     #CmdRstTrueTime;
      =     #CmdRstFalseTime;
      =     #CmdRunTimeoutTime;
      AN    #InPreAlarmTrue;	//[3.0]
      R     #OutPreAlarmTrue;	//[3.0]
      AN    #InPreAlarmFalse;	//[3.0]
      R     #OutPreAlarmFalse;	//[3.0]
//===Set Output fault reset
      A     "GCS7_Gr_OutTick1s";	// Gr.OutTick1s [3.5] [4.2]
      AN    #StFault;	//[3.2]
      R     #OutpFaultReset;	//[3.3]
      AN    #InMonTrue;	//[4.5]
      AN    #InMonFalse;	//[4.5]
      O     #StFault;	//[3.2]
      O     #tmpLocal;	//[3.5]
      A     "GCS7_Gr_OutTick1s";	// Gr.OutTick1s [3.1]
      A     #CmdFaultReset;
      S     #OutpFaultReset;
      A     "GCS7_Gr_OutTick1s";	// Gr.OutTick1s [3.5]
      R     #CmdFaultReset;
//--Output for group 
      AN    #InLocal;
      A     #InDPFault;
      S     "GCS7_Gr_InDPFault";
      AN    #InLocal;
      A     #InHWStop;
      S     "GCS7_Gr_InHWStop";
NETWORK
TITLE = State Code
      A     #InLocal;	// [3.0]
      JCN   STC1;
      A     #InpFaultDev;	// [3.0]
      AN    #InpTrue;	// [4.0]
      L     61;	// [3.0]
      JC    STC9;	//Code StFalse.FaultDev
      A     #InpFaultDev;	// [3.0]
      A     #InpTrue;	// [4.0]
      L     63;	// [3.0]
      JC    STC9;	//Code StTrue.FaultDev
//--------------------
STC1: AN    #StFalse;
      JC    STC2;
      L     41;	//Code: StFalse.HWStop
      A     #InHWStop;
      JC    STC9;
      L     51;	//Code: StFalse.DPFault
      A     #InDPFault;
      JC    STC9;
      L     1;	//Code: StFalse
      JU    STC8;
//--------------------
STC2: A     #StCtoTrue;
      L     2;	//Code: StCtoTrue
      JC    STC8;
//--------------------
      AN    #StTrue;
      JC    STC4;
      L     43;	//Code: StTrue.HWStop
      A     #InHWStop;
      JC    STC9;
      L     53;	//Code: StTrue.DPFault
      A     #InDPFault;
      JC    STC9;
      L     3;	//Code: StTrue
      JC    STC8;
//--------------------
STC4: A     #StCtoFalse;
      L     4;	// Code: StCtoFalse
      JC    STC8;
      A     #InpFaultDev;	// [3.0]
      L     31;	// [3.0]
      JC    STC9;	// [3.0]
      L     32;	// Code: fault
      JU    STC9;
      AN    #OutPreAlarmTrue;
      JC    STC9;
STC8: AN    #OutPreAlarmFalse;	// Code: StXx.Warning [3.0]
      AN    #OutPreAlarmTrue;	// Code: StXx.Warning [3.0]
      JC    STC9;	// Code: StXx.Warning [3.0]
      +     10;	// Code: StXx.Warning [3.0] =+10
STC9: L     #StCode;	// Old state code
      TAK;
      T     #StCode;	// Save state code
      <>I;
      L     3;	// Load code for CBit methode
      CC    "SYS_CBitCtrl";
END_FUNCTION_BLOCK

